LIN {X 0,Y 284.997,Z 899.013,A -85,B 0,C 180,E1 -17446.451,E2 -17446.451} C_VEL
LIN {X 0,Y 283.143,Z 901.991,A -85,B 0,C 180,E1 -17448.547,E2 -17448.547} C_VEL
LIN {X 0,Y 282.042,Z 903.588,A -85,B 0,C 180,E1 -17449.955,E2 -17449.955} C_VEL
LIN {X 0,Y 280.982,Z 904.651,A -85,B 0,C 180,E1 -17451.369,E2 -17451.369} C_VEL
LIN {X 0,Y 279.65,Z 905.657,A -85,B 0,C 180,E1 -17454.231,E2 -17454.231} C_VEL
LIN {X 0,Y 278.605,Z 905.018,A -85,B 0,C 180,E1 -17457.108,E2 -17457.108} C_VEL
LIN {X 0,Y 278.2,Z 904.125,A -85,B 0,C 180,E1 -17458.552,E2 -17458.552} C_VEL
LIN {X 0,Y 277.742,Z 902.734,A -85,B 0,C 180,E1 -17460,E2 -17460} C_VEL
LIN {X 0,Y 277.629,Z 899.945,A -85,B 0,C 180,E1 -17462.176,E2 -17462.176} C_VEL
LIN {X 0,Y 277.371,Z 896.204,A -85,B 0,C 180,E1 -17464.36,E2 -17464.36} C_VEL
LIN {X 0,Y 277.84,Z 891.35,A -85,B 0,C 180,E1 -17466.536,E2 -17466.536} C_VEL
LIN {X 0,Y 278.22,Z 885.341,A -85,B 0,C 180,E1 -17468.718,E2 -17468.718} C_VEL
LIN {X 0,Y 278.889,Z 876.721,A -85,B 0,C 180,E1 -17471.226,E2 -17471.226} C_VEL
LIN {X 0,Y 279.577,Z 868.835,A -85,B 0,C 180,E1 -17473.076,E2 -17473.076} C_VEL
LIN {X 0,Y 280.358,Z 859.638,A -85,B 0,C 180,E1 -17474.889,E2 -17474.889} C_VEL
LIN {X 0,Y 281.096,Z 850.958,A -85,B 0,C 180,E1 -17476.336,E2 -17476.336} C_VEL
LIN {X 0,Y 282.024,Z 840.057,A -85,B 0,C 180,E1 -17477.875,E2 -17477.875} C_VEL
LIN {X 0,Y 281.926,Z 836.631,A -85,B 0,C 180,E1 -17478.309,E2 -17478.309} C_VEL
LIN {X 0,Y 278.815,Z 824.242,A -85,B 0,C 180,E1 -17479.779,E2 -17479.779} C_VEL
LIN {X 0,Y 277.294,Z 817.935,A -85,B 0,C 180,E1 -17480.464,E2 -17480.464} C_VEL
LIN {X 0,Y 277.243,Z 817.949,A -85,B 0,C 180,E1 -17484.131,E2 -17484.131} C_VEL
LIN {X 0,Y 277.242,Z 817.938,A -85,B 0,C 180,E1 -17487.468,E2 -17487.468} C_VEL
LIN {X 0,Y 277.236,Z 817.947,A -85,B 0,C 180,E1 -17490.465,E2 -17490.465} C_VEL
LIN {X 0,Y 277.253,Z 817.94,A -85,B 0,C 180,E1 -17493.895,E2 -17493.895} C_VEL
LIN {X 0,Y 277.258,Z 817.939,A -85,B 0,C 180,E1 -17497.471,E2 -17497.471} C_VEL
LIN {X 0,Y 277.191,Z 817.953,A -85,B 0,C 180,E1 -17501.24,E2 -17501.24} C_VEL
LIN {X 0,Y 277.181,Z 817.956,A -85,B 0,C 180,E1 -17505.231,E2 -17505.231} C_VEL
LIN {X 0,Y 277.184,Z 817.956,A -85,B 0,C 180,E1 -17508.756,E2 -17508.756} C_VEL
LIN {X 0,Y 277.255,Z 817.945,A -85,B 0,C 180,E1 -17512.526,E2 -17512.526} C_VEL
LIN {X 0,Y 277.253,Z 817.95,A -85,B 0,C 180,E1 -17516.103,E2 -17516.103} C_VEL
LIN {X 0,Y 277.268,Z 817.941,A -85,B 0,C 180,E1 -17519.537,E2 -17519.537} C_VEL
LIN {X 0,Y 277.349,Z 817.93,A -85,B 0,C 180,E1 -17523.673,E2 -17523.673} C_VEL
LIN {X 0,Y 277.358,Z 817.943,A -85,B 0,C 180,E1 -17524.356,E2 -17524.356} C_VEL
LIN {X 0,Y 278.289,Z 820.641,A -85,B 0,C 180,E1 -17524.651,E2 -17524.651} C_VEL
LIN {X 0,Y 282.727,Z 831.715,A -85,B 0,C 180,E1 -17526.103,E2 -17526.103} C_VEL
LIN {X 0,Y 285.992,Z 841.823,A -85,B 0,C 180,E1 -17527.586,E2 -17527.586} C_VEL
LIN {X 0,Y 287.967,Z 848.891,A -85,B 0,C 180,E1 -17528.746,E2 -17528.746} C_VEL
LIN {X 0,Y 287.007,Z 857.045,A -85,B 0,C 180,E1 -17529.949,E2 -17529.949} C_VEL
LIN {X 0,Y 285.466,Z 866.858,A -85,B 0,C 180,E1 -17531.703,E2 -17531.703} C_VEL
LIN {X 0,Y 283.92,Z 874.9,A -85,B 0,C 180,E1 -17533.459,E2 -17533.459} C_VEL
LIN {X 0,Y 282.324,Z 882.758,A -85,B 0,C 180,E1 -17535.583,E2 -17535.583} C_VEL
LIN {X 0,Y 281.178,Z 889.027,A -85,B 0,C 180,E1 -17537.731,E2 -17537.731} C_VEL
LIN {X 0,Y 280.049,Z 894.02,A -85,B 0,C 180,E1 -17539.88,E2 -17539.88} C_VEL
LIN {X 0,Y 278.971,Z 897.914,A -85,B 0,C 180,E1 -17542.033,E2 -17542.033} C_VEL
LIN {X 0,Y 278.316,Z 900.764,A -85,B 0,C 180,E1 -17544.2,E2 -17544.2} C_VEL
LIN {X 0,Y 278.247,Z 902.093,A -85,B 0,C 180,E1 -17545.652,E2 -17545.652} C_VEL
LIN {X 0,Y 277.82,Z 903.673,A -85,B 0,C 180,E1 -17548.548,E2 -17548.548} C_VEL
LIN {X 0,Y 277.759,Z 903.902,A -85,B 0,C 180,E1 -17549.997,E2 -17549.997} C_VEL
LIN {X 0,Y 278.009,Z 903.133,A -85,B 0,C 180,E1 -17552.895,E2 -17552.895} C_VEL
LIN {X 0,Y 278.229,Z 902.189,A -85,B 0,C 180,E1 -17554.343,E2 -17554.343} C_VEL
LIN {X 0,Y 278.302,Z 900.9,A -85,B 0,C 180,E1 -17555.795,E2 -17555.795} C_VEL
LIN {X 0,Y 278.957,Z 898.092,A -85,B 0,C 180,E1 -17557.962,E2 -17557.962} C_VEL
LIN {X 0,Y 280.065,Z 894.248,A -85,B 0,C 180,E1 -17560.114,E2 -17560.114} C_VEL
LIN {X 0,Y 281.138,Z 889.336,A -85,B 0,C 180,E1 -17562.265,E2 -17562.265} C_VEL
LIN {X 0,Y 282.293,Z 883.16,A -85,B 0,C 180,E1 -17564.413,E2 -17564.413} C_VEL
LIN {X 0,Y 283.869,Z 875.385,A -85,B 0,C 180,E1 -17566.539,E2 -17566.539} C_VEL
LIN {X 0,Y 285.315,Z 867.455,A -85,B 0,C 180,E1 -17568.301,E2 -17568.301} C_VEL
LIN {X 0,Y 286.932,Z 857.756,A -85,B 0,C 180,E1 -17570.051,E2 -17570.051} C_VEL
LIN {X 0,Y 288.057,Z 849.407,A -85,B 0,C 180,E1 -17571.287,E2 -17571.287} C_VEL
LIN {X 0,Y 285.703,Z 840.645,A -85,B 0,C 180,E1 -17572.712,E2 -17572.712} C_VEL
LIN {X 0,Y 282.328,Z 830.734,A -85,B 0,C 180,E1 -17574.161,E2 -17574.161} C_VEL
LIN {X 0,Y 278.161,Z 820.468,A -85,B 0,C 180,E1 -17575.5,E2 -17575.5} C_VEL
LIN {X 0,Y 277.347,Z 817.939,A -85,B 0,C 180,E1 -17575.816,E2 -17575.816} C_VEL
LIN {X 0,Y 277.284,Z 817.946,A -85,B 0,C 180,E1 -17578.785,E2 -17578.785} C_VEL
LIN {X 0,Y 277.249,Z 817.95,A -85,B 0,C 180,E1 -17583.225,E2 -17583.225} C_VEL
LIN {X 0,Y 277.319,Z 817.944,A -85,B 0,C 180,E1 -17585.809,E2 -17585.809} C_VEL
LIN {X 0,Y 277.26,Z 817.948,A -85,B 0,C 180,E1 -17589.32,E2 -17589.32} C_VEL
LIN {X 0,Y 277.277,Z 817.945,A -85,B 0,C 180,E1 -17593.181,E2 -17593.181} C_VEL
LIN {X 0,Y 277.271,Z 817.939,A -85,B 0,C 180,E1 -17597.308,E2 -17597.308} C_VEL
LIN {X 0,Y 277.267,Z 817.942,A -85,B 0,C 180,E1 -17600.677,E2 -17600.677} C_VEL
LIN {X 0,Y 277.294,Z 817.943,A -85,B 0,C 180,E1 -17604.343,E2 -17604.343} C_VEL
LIN {X 0,Y 277.232,Z 817.95,A -85,B 0,C 180,E1 -17607.835,E2 -17607.835} C_VEL
LIN {X 0,Y 277.276,Z 817.946,A -85,B 0,C 180,E1 -17611.211,E2 -17611.211} C_VEL
LIN {X 0,Y 277.3,Z 817.937,A -85,B 0,C 180,E1 -17614.478,E2 -17614.478} C_VEL
LIN {X 0,Y 277.271,Z 817.944,A -85,B 0,C 180,E1 -17617.653,E2 -17617.653} C_VEL
LIN {X 0,Y 277.33,Z 817.937,A -85,B 0,C 180,E1 -17620.765,E2 -17620.765} C_VEL
LIN {X 0,Y 277.42,Z 817.92,A -85,B 0,C 180,E1 -17625.325,E2 -17625.325} C_VEL
LIN {X 0,Y 277.492,Z 817.914,A -85,B 0,C 180,E1 -17629.788,E2 -17629.788} C_VEL
LIN {X 0,Y 277.633,Z 817.902,A -85,B 0,C 180,E1 -17632.728,E2 -17632.728} C_VEL
LIN {X 0,Y 277.806,Z 817.881,A -85,B 0,C 180,E1 -17638.55,E2 -17638.55} C_VEL
LIN {X 0,Y 277.805,Z 817.884,A -85,B 0,C 180,E1 -17641.45,E2 -17641.45} C_VEL
LIN {X 0,Y 277.624,Z 817.903,A -85,B 0,C 180,E1 -17647.272,E2 -17647.272} C_VEL
LIN {X 0,Y 277.607,Z 817.904,A -85,B 0,C 180,E1 -17649.053,E2 -17649.053} C_VEL
LIN {X 0,Y 276.969,Z 817.986,A -85,B 0,C 180,E1 -17650.262,E2 -17650.262} C_VEL
LIN {X 0,Y 274.06,Z 818.349,A -85,B 0,C 180,E1 -17652.228,E2 -17652.228} C_VEL
LIN {X 0,Y 271.554,Z 818.659,A -85,B 0,C 180,E1 -17653.826,E2 -17653.826} C_VEL
LIN {X 0,Y 270.464,Z 818.795,A -85,B 0,C 180,E1 -17655.068,E2 -17655.068} C_VEL
LIN {X 0,Y 270.369,Z 818.807,A -85,B 0,C 180,E1 -17655.489,E2 -17655.489} C_VEL
LIN {X 0,Y 270.285,Z 818.819,A -85,B 0,C 180,E1 -17659.757,E2 -17659.757} C_VEL
LIN {X 0,Y 270.209,Z 818.826,A -85,B 0,C 180,E1 -17664.592,E2 -17664.592} C_VEL
LIN {X 0,Y 270.184,Z 818.825,A -85,B 0,C 180,E1 -17667.918,E2 -17667.918} C_VEL
LIN {X 0,Y 270.16,Z 818.833,A -85,B 0,C 180,E1 -17671.351,E2 -17671.351} C_VEL
LIN {X 0,Y 270.211,Z 818.827,A -85,B 0,C 180,E1 -17675.588,E2 -17675.588} C_VEL
LIN {X 0,Y 270.226,Z 818.92,A -85,B 0,C 180,E1 -17676.275,E2 -17676.275} C_VEL
LIN {X 0,Y 271.583,Z 825.509,A -85,B 0,C 180,E1 -17680.312,E2 -17680.312} C_VEL
LIN {X 0,Y 272.964,Z 832.072,A -85,B 0,C 180,E1 -17684.041,E2 -17684.041} C_VEL
LIN {X 0,Y 274.469,Z 840.068,A -85,B 0,C 180,E1 -17688.264,E2 -17688.264} C_VEL
LIN {X 0,Y 275.333,Z 845.207,A -85,B 0,C 180,E1 -17690.824,E2 -17690.824} C_VEL
LIN {X 0,Y 274.944,Z 848.645,A -85,B 0,C 180,E1 -17692.411,E2 -17692.411} C_VEL
LIN {X 0,Y 273.277,Z 857.605,A -85,B 0,C 180,E1 -17696.436,E2 -17696.436} C_VEL
LIN {X 0,Y 271.582,Z 868.258,A -85,B 0,C 180,E1 -17701.195,E2 -17701.195} C_VEL
LIN {X 0,Y 271.138,Z 871.591,A -85,B 0,C 180,E1 -17702.697,E2 -17702.697} C_VEL
LIN {X 0,Y 273.513,Z 886.239,A -85,B 0,C 180,E1 -17703.606,E2 -17703.606} C_VEL
LIN {X 0,Y 274.931,Z 899.031,A -85,B 0,C 180,E1 -17704.641,E2 -17704.641} C_VEL
LIN {X 0,Y 275.523,Z 911.781,A -85,B 0,C 180,E1 -17705.916,E2 -17705.916} C_VEL
LIN {X 0,Y 275.466,Z 923.215,A -85,B 0,C 180,E1 -17707.312,E2 -17707.312} C_VEL
LIN {X 0,Y 274.898,Z 933.568,A -85,B 0,C 180,E1 -17708.834,E2 -17708.834} C_VEL
LIN {X 0,Y 274.438,Z 941.169,A -85,B 0,C 180,E1 -17710.168,E2 -17710.168} C_VEL
LIN {X 0,Y 272.711,Z 950.162,A -85,B 0,C 180,E1 -17711.989,E2 -17711.989} C_VEL
LIN {X 0,Y 271.023,Z 958.971,A -85,B 0,C 180,E1 -17714.203,E2 -17714.203} C_VEL
LIN {X 0,Y 270.056,Z 966.097,A -85,B 0,C 180,E1 -17716.457,E2 -17716.457} C_VEL
LIN {X 0,Y 269.414,Z 971.84,A -85,B 0,C 180,E1 -17718.72,E2 -17718.72} C_VEL
LIN {X 0,Y 269.186,Z 976.397,A -85,B 0,C 180,E1 -17720.99,E2 -17720.99} C_VEL
LIN {X 0,Y 269.222,Z 979.193,A -85,B 0,C 180,E1 -17722.741,E2 -17722.741} C_VEL
LIN {X 0,Y 269.55,Z 982.334,A -85,B 0,C 180,E1 -17725.517,E2 -17725.517} C_VEL
LIN {X 0,Y 269.706,Z 983.411,A -85,B 0,C 180,E1 -17727.015,E2 -17727.015} C_VEL
LIN {X 0,Y 269.852,Z 984.074,A -85,B 0,C 180,E1 -17728.51,E2 -17728.51} C_VEL
LIN {X 0,Y 269.995,Z 984.319,A -85,B 0,C 180,E1 -17730.003,E2 -17730.003} C_VEL
LIN {X 0,Y 269.853,Z 984.064,A -85,B 0,C 180,E1 -17731.495,E2 -17731.495} C_VEL
LIN {X 0,Y 269.71,Z 983.395,A -85,B 0,C 180,E1 -17732.99,E2 -17732.99} C_VEL
LIN {X 0,Y 269.575,Z 982.315,A -85,B 0,C 180,E1 -17734.488,E2 -17734.488} C_VEL
LIN {X 0,Y 269.238,Z 979.122,A -85,B 0,C 180,E1 -17737.284,E2 -17737.284} C_VEL
LIN {X 0,Y 269.529,Z 971.343,A -85,B 0,C 180,E1 -17742.043,E2 -17742.043} C_VEL
LIN {X 0,Y 270.381,Z 966.739,A -85,B 0,C 180,E1 -17744.299,E2 -17744.299} C_VEL
LIN {X 0,Y 271.681,Z 961.017,A -85,B 0,C 180,E1 -17746.535,E2 -17746.535} C_VEL
LIN {X 0,Y 273.549,Z 954.239,A -85,B 0,C 180,E1 -17748.735,E2 -17748.735} C_VEL
LIN {X 0,Y 275.991,Z 946.224,A -85,B 0,C 180,E1 -17750.888,E2 -17750.888} C_VEL
LIN {X 0,Y 277.399,Z 940.261,A -85,B 0,C 180,E1 -17752.338,E2 -17752.338} C_VEL
LIN {X 0,Y 279.567,Z 929.919,A -85,B 0,C 180,E1 -17754.509,E2 -17754.509} C_VEL
LIN {X 0,Y 281.86,Z 919.067,A -85,B 0,C 180,E1 -17756.455,E2 -17756.455} C_VEL
LIN {X 0,Y 282.915,Z 909.244,A -85,B 0,C 180,E1 -17758.166,E2 -17758.166} C_VEL
LIN {X 0,Y 283.359,Z 896.995,A -85,B 0,C 180,E1 -17760.265,E2 -17760.265} C_VEL
LIN {X 0,Y 283.177,Z 886.629,A -85,B 0,C 180,E1 -17762.084,E2 -17762.084} C_VEL
LIN {X 0,Y 282.457,Z 875.054,A -85,B 0,C 180,E1 -17764.252,E2 -17764.252} C_VEL
LIN {X 0,Y 281.688,Z 866.988,A -85,B 0,C 180,E1 -17765.899,E2 -17765.899} C_VEL
LIN {X 0,Y 281.166,Z 861.203,A -85,B 0,C 180,E1 -17767.187,E2 -17767.187} C_VEL
LIN {X 0,Y 281.146,Z 859.94,A -85,B 0,C 180,E1 -17767.42,E2 -17767.42} C_VEL
LIN {X 0,Y 279.903,Z 851.044,A -85,B 0,C 180,E1 -17769.942,E2 -17769.942} C_VEL
LIN {X 0,Y 279.125,Z 846.061,A -85,B 0,C 180,E1 -17771.937,E2 -17771.937} C_VEL
LIN {X 0,Y 278.623,Z 842.393,A -85,B 0,C 180,E1 -17773.993,E2 -17773.993} C_VEL
LIN {X 0,Y 278.659,Z 839.748,A -85,B 0,C 180,E1 -17776.004,E2 -17776.004} C_VEL
LIN {X 0,Y 278.898,Z 838.691,A -85,B 0,C 180,E1 -17777.127,E2 -17777.127} C_VEL
LIN {X 0,Y 279.657,Z 837.646,A -85,B 0,C 180,E1 -17779.201,E2 -17779.201} C_VEL
LIN {X 0,Y 280.989,Z 837.503,A -85,B 0,C 180,E1 -17781.296,E2 -17781.296} C_VEL
LIN {X 0,Y 282.724,Z 838.756,A -85,B 0,C 180,E1 -17783.373,E2 -17783.373} C_VEL
LIN {X 0,Y 284.775,Z 840.777,A -85,B 0,C 180,E1 -17785.415,E2 -17785.415} C_VEL
LIN {X 0,Y 287.225,Z 843.725,A -85,B 0,C 180,E1 -17787.431,E2 -17787.431} C_VEL
LIN {X 0,Y 290.331,Z 851.625,A -85,B 0,C 180,E1 -17790.631,E2 -17790.631} C_VEL
LIN {X 0,Y 292.153,Z 858.072,A -85,B 0,C 180,E1 -17792.802,E2 -17792.802} C_VEL
LIN {X 0,Y 293.327,Z 864.655,A -85,B 0,C 180,E1 -17794.831,E2 -17794.831} C_VEL
LIN {X 0,Y 293.448,Z 865.932,A -85,B 0,C 180,E1 -17795.221,E2 -17795.221} C_VEL
LIN {X 0,Y 291.978,Z 870.915,A -85,B 0,C 180,E1 -17796.185,E2 -17796.185} C_VEL
LIN {X 0,Y 288.671,Z 879.706,A -85,B 0,C 180,E1 -17798.129,E2 -17798.129} C_VEL
LIN {X 0,Y 285.979,Z 886.069,A -85,B 0,C 180,E1 -17799.876,E2 -17799.876} C_VEL
LIN {X 0,Y 284.047,Z 890.377,A -85,B 0,C 180,E1 -17801.237,E2 -17801.237} C_VEL
LIN {X 0,Y 281.48,Z 895.633,A -85,B 0,C 180,E1 -17803.314,E2 -17803.314} C_VEL
LIN {X 0,Y 279.135,Z 899.868,A -85,B 0,C 180,E1 -17805.417,E2 -17805.417} C_VEL
LIN {X 0,Y 277.722,Z 902.115,A -85,B 0,C 180,E1 -17806.835,E2 -17806.835} C_VEL
LIN {X 0,Y 275.261,Z 905.236,A -85,B 0,C 180,E1 -17809.705,E2 -17809.705} C_VEL
LIN {X 0,Y 274.166,Z 906.273,A -85,B 0,C 180,E1 -17811.153,E2 -17811.153} C_VEL
LIN {X 0,Y 272.71,Z 906.976,A -85,B 0,C 180,E1 -17814.083,E2 -17814.083} C_VEL
LIN {X 0,Y 272.154,Z 906.742,A -85,B 0,C 180,E1 -17815.557,E2 -17815.557} C_VEL
LIN {X 0,Y 271.615,Z 906.142,A -85,B 0,C 180,E1 -17817.034,E2 -17817.034} C_VEL
LIN {X 0,Y 271.188,Z 905.089,A -85,B 0,C 180,E1 -17818.515,E2 -17818.515} C_VEL
LIN {X 0,Y 270.715,Z 903.642,A -85,B 0,C 180,E1 -17820,E2 -17820} C_VEL
LIN {X 0,Y 270.594,Z 900.68,A -85,B 0,C 180,E1 -17822.233,E2 -17822.233} C_VEL
LIN {X 0,Y 270.333,Z 896.764,A -85,B 0,C 180,E1 -17824.473,E2 -17824.473} C_VEL
LIN {X 0,Y 270.798,Z 891.735,A -85,B 0,C 180,E1 -17826.707,E2 -17826.707} C_VEL
LIN {X 0,Y 271.322,Z 883.824,A -85,B 0,C 180,E1 -17829.462,E2 -17829.462} C_VEL
LIN {X 0,Y 271.916,Z 876.431,A -85,B 0,C 180,E1 -17831.555,E2 -17831.555} C_VEL
LIN {X 0,Y 272.631,Z 868.408,A -85,B 0,C 180,E1 -17833.415,E2 -17833.415} C_VEL
LIN {X 0,Y 273.356,Z 859.973,A -85,B 0,C 180,E1 -17835.089,E2 -17835.089} C_VEL
LIN {X 0,Y 274.112,Z 851.176,A -85,B 0,C 180,E1 -17836.573,E2 -17836.573} C_VEL
LIN {X 0,Y 275.005,Z 840.836,A -85,B 0,C 180,E1 -17838.057,E2 -17838.057} C_VEL
LIN {X 0,Y 275.02,Z 838.204,A -85,B 0,C 180,E1 -17838.396,E2 -17838.396} C_VEL
LIN {X 0,Y 271.851,Z 825.586,A -85,B 0,C 180,E1 -17839.946,E2 -17839.946} C_VEL
LIN {X 0,Y 270.24,Z 818.813,A -85,B 0,C 180,E1 -17840.679,E2 -17840.679} C_VEL
LIN {X 0,Y 270.185,Z 818.827,A -85,B 0,C 180,E1 -17844.594,E2 -17844.594} C_VEL
LIN {X 0,Y 270.192,Z 818.818,A -85,B 0,C 180,E1 -17847.918,E2 -17847.918} C_VEL
LIN {X 0,Y 270.177,Z 818.826,A -85,B 0,C 180,E1 -17851.349,E2 -17851.349} C_VEL
LIN {X 0,Y 270.205,Z 818.823,A -85,B 0,C 180,E1 -17854.905,E2 -17854.905} C_VEL
LIN {X 0,Y 270.206,Z 818.822,A -85,B 0,C 180,E1 -17858.709,E2 -17858.709} C_VEL
LIN {X 0,Y 270.156,Z 818.828,A -85,B 0,C 180,E1 -17863.244,E2 -17863.244} C_VEL
LIN {X 0,Y 270.158,Z 818.83,A -85,B 0,C 180,E1 -17867.436,E2 -17867.436} C_VEL
LIN {X 0,Y 270.173,Z 818.831,A -85,B 0,C 180,E1 -17871.366,E2 -17871.366} C_VEL
LIN {X 0,Y 270.205,Z 818.825,A -85,B 0,C 180,E1 -17875.092,E2 -17875.092} C_VEL
LIN {X 0,Y 270.207,Z 818.82,A -85,B 0,C 180,E1 -17879.129,E2 -17879.129} C_VEL
LIN {X 0,Y 270.307,Z 818.807,A -85,B 0,C 180,E1 -17883.61,E2 -17883.61} C_VEL
LIN {X 0,Y 270.881,Z 820.853,A -85,B 0,C 180,E1 -17883.826,E2 -17883.826} C_VEL
LIN {X 0,Y 275.054,Z 830.761,A -85,B 0,C 180,E1 -17885.164,E2 -17885.164} C_VEL
LIN {X 0,Y 278.475,Z 840.628,A -85,B 0,C 180,E1 -17886.638,E2 -17886.638} C_VEL
LIN {X 0,Y 281.211,Z 850.251,A -85,B 0,C 180,E1 -17888.255,E2 -17888.255} C_VEL
LIN {X 0,Y 281.158,Z 853.471,A -85,B 0,C 180,E1 -17888.749,E2 -17888.749} C_VEL
LIN {X 0,Y 279.711,Z 862.284,A -85,B 0,C 180,E1 -17890.169,E2 -17890.169} C_VEL
LIN {X 0,Y 278.168,Z 871.306,A -85,B 0,C 180,E1 -17891.968,E2 -17891.968} C_VEL
LIN {X 0,Y 276.276,Z 880.085,A -85,B 0,C 180,E1 -17894.127,E2 -17894.127} C_VEL
LIN {X 0,Y 274.95,Z 886.884,A -85,B 0,C 180,E1 -17896.246,E2 -17896.246} C_VEL
LIN {X 0,Y 273.976,Z 891.821,A -85,B 0,C 180,E1 -17898.155,E2 -17898.155} C_VEL
LIN {X 0,Y 272.659,Z 896.459,A -85,B 0,C 180,E1 -17900.352,E2 -17900.352} C_VEL
LIN {X 0,Y 271.763,Z 899.981,A -85,B 0,C 180,E1 -17902.568,E2 -17902.568} C_VEL
LIN {X 0,Y 271.328,Z 901.796,A -85,B 0,C 180,E1 -17904.05,E2 -17904.05} C_VEL
LIN {X 0,Y 271.244,Z 903.125,A -85,B 0,C 180,E1 -17905.539,E2 -17905.539} C_VEL
LIN {X 0,Y 270.798,Z 904.704,A -85,B 0,C 180,E1 -17908.51,E2 -17908.51} C_VEL
LIN {X 0,Y 270.735,Z 904.933,A -85,B 0,C 180,E1 -17909.997,E2 -17909.997} C_VEL
LIN {X 0,Y 270.995,Z 904.163,A -85,B 0,C 180,E1 -17912.97,E2 -17912.97} C_VEL
LIN {X 0,Y 271.228,Z 903.22,A -85,B 0,C 180,E1 -17914.456,E2 -17914.456} C_VEL
LIN {X 0,Y 271.314,Z 901.93,A -85,B 0,C 180,E1 -17915.945,E2 -17915.945} C_VEL
LIN {X 0,Y 272.002,Z 899.123,A -85,B 0,C 180,E1 -17918.167,E2 -17918.167} C_VEL
LIN {X 0,Y 273.152,Z 895.278,A -85,B 0,C 180,E1 -17920.373,E2 -17920.373} C_VEL
LIN {X 0,Y 274.281,Z 890.365,A -85,B 0,C 180,E1 -17922.577,E2 -17922.577} C_VEL
LIN {X 0,Y 275.496,Z 884.189,A -85,B 0,C 180,E1 -17924.777,E2 -17924.777} C_VEL
LIN {X 0,Y 277.142,Z 876.414,A -85,B 0,C 180,E1 -17926.952,E2 -17926.952} C_VEL
LIN {X 0,Y 278.666,Z 868.481,A -85,B 0,C 180,E1 -17928.754,E2 -17928.754} C_VEL
LIN {X 0,Y 280.349,Z 858.783,A -85,B 0,C 180,E1 -17930.543,E2 -17930.543} C_VEL
LIN {X 0,Y 281.375,Z 852.217,A -85,B 0,C 180,E1 -17931.545,E2 -17931.545} C_VEL
LIN {X 0,Y 280.804,Z 848.504,A -85,B 0,C 180,E1 -17932.174,E2 -17932.174} C_VEL
LIN {X 0,Y 277.633,Z 837.999,A -85,B 0,C 180,E1 -17933.889,E2 -17933.889} C_VEL
LIN {X 0,Y 273.945,Z 827.91,A -85,B 0,C 180,E1 -17935.351,E2 -17935.351} C_VEL
LIN {X 0,Y 270.36,Z 819.221,A -85,B 0,C 180,E1 -17936.476,E2 -17936.476} C_VEL
LIN {X 0,Y 270.304,Z 818.816,A -85,B 0,C 180,E1 -17936.54,E2 -17936.54} C_VEL
LIN {X 0,Y 270.195,Z 818.829,A -85,B 0,C 180,E1 -17940.867,E2 -17940.867} C_VEL
LIN {X 0,Y 270.209,Z 818.827,A -85,B 0,C 180,E1 -17944.901,E2 -17944.901} C_VEL
LIN {X 0,Y 270.214,Z 818.827,A -85,B 0,C 180,E1 -17948.714,E2 -17948.714} C_VEL
LIN {X 0,Y 270.253,Z 818.822,A -85,B 0,C 180,E1 -17952.538,E2 -17952.538} C_VEL
LIN {X 0,Y 270.223,Z 818.82,A -85,B 0,C 180,E1 -17956.733,E2 -17956.733} C_VEL
LIN {X 0,Y 270.254,Z 818.82,A -85,B 0,C 180,E1 -17959.448,E2 -17959.448} C_VEL
LIN {X 0,Y 270.247,Z 818.82,A -85,B 0,C 180,E1 -17963.719,E2 -17963.719} C_VEL
LIN {X 0,Y 270.192,Z 818.828,A -85,B 0,C 180,E1 -17966.891,E2 -17966.891} C_VEL
LIN {X 0,Y 270.216,Z 818.819,A -85,B 0,C 180,E1 -17970.385,E2 -17970.385} C_VEL
LIN {X 0,Y 270.25,Z 818.816,A -85,B 0,C 180,E1 -17973.762,E2 -17973.762} C_VEL
LIN {X 0,Y 270.219,Z 818.826,A -85,B 0,C 180,E1 -17977.037,E2 -17977.037} C_VEL
LIN {X 0,Y 270.287,Z 818.812,A -85,B 0,C 180,E1 -17980.243,E2 -17980.243} C_VEL
LIN {X 0,Y 270.388,Z 818.794,A -85,B 0,C 180,E1 -17984.934,E2 -17984.934} C_VEL
LIN {X 0,Y 270.427,Z 818.795,A -85,B 0,C 180,E1 -17989.518,E2 -17989.518} C_VEL
LIN {X 0,Y 270.592,Z 818.778,A -85,B 0,C 180,E1 -17992.538,E2 -17992.538} C_VEL
LIN {X 0,Y 270.772,Z 818.758,A -85,B 0,C 180,E1 -17998.513,E2 -17998.513} C_VEL
LIN {X 0,Y 270.77,Z 818.761,A -85,B 0,C 180,E1 -18001.487,E2 -18001.487} C_VEL
LIN {X 0,Y 270.584,Z 818.781,A -85,B 0,C 180,E1 -18007.462,E2 -18007.462} C_VEL
LIN {X 0,Y 270.426,Z 818.798,A -85,B 0,C 180,E1 -18010.482,E2 -18010.482} C_VEL
LIN {X 0,Y 270.369,Z 818.807,A -85,B 0,C 180,E1 -18015.489,E2 -18015.489} C_VEL
LIN {X 0,Y 269.677,Z 818.896,A -85,B 0,C 180,E1 -18016.731,E2 -18016.731} C_VEL
LIN {X 0,Y 266.778,Z 819.263,A -85,B 0,C 180,E1 -18018.753,E2 -18018.753} C_VEL
LIN {X 0,Y 264.307,Z 819.571,A -85,B 0,C 180,E1 -18020.397,E2 -18020.397} C_VEL
LIN {X 0,Y 263.221,Z 819.701,A -85,B 0,C 180,E1 -18021.673,E2 -18021.673} C_VEL
LIN {X 0,Y 263.118,Z 819.71,A -85,B 0,C 180,E1 -18022.106,E2 -18022.106} C_VEL
LIN {X 0,Y 263.153,Z 819.704,A -85,B 0,C 180,E1 -18025.297,E2 -18025.297} C_VEL
LIN {X 0,Y 263.119,Z 819.712,A -85,B 0,C 180,E1 -18028.737,E2 -18028.737} C_VEL
LIN {X 0,Y 263.114,Z 819.708,A -85,B 0,C 180,E1 -18032.291,E2 -18032.291} C_VEL
LIN {X 0,Y 263.196,Z 819.769,A -85,B 0,C 180,E1 -18035.506,E2 -18035.506} C_VEL
LIN {X 0,Y 264.498,Z 826.24,A -85,B 0,C 180,E1 -18039.621,E2 -18039.621} C_VEL
LIN {X 0,Y 265.833,Z 832.682,A -85,B 0,C 180,E1 -18043.423,E2 -18043.423} C_VEL
LIN {X 0,Y 267.239,Z 840.004,A -85,B 0,C 180,E1 -18047.422,E2 -18047.422} C_VEL
LIN {X 0,Y 268.223,Z 845.529,A -85,B 0,C 180,E1 -18050.307,E2 -18050.307} C_VEL
LIN {X 0,Y 268.367,Z 847.054,A -85,B 0,C 180,E1 -18051.064,E2 -18051.064} C_VEL
LIN {X 0,Y 266.939,Z 854.856,A -85,B 0,C 180,E1 -18054.704,E2 -18054.704} C_VEL
LIN {X 0,Y 264.953,Z 865.764,A -85,B 0,C 180,E1 -18059.74,E2 -18059.74} C_VEL
LIN {X 0,Y 264.257,Z 870.498,A -85,B 0,C 180,E1 -18061.93,E2 -18061.93} C_VEL
LIN {X 0,Y 266.677,Z 885.004,A -85,B 0,C 180,E1 -18062.868,E2 -18062.868} C_VEL
LIN {X 0,Y 268.111,Z 897.835,A -85,B 0,C 180,E1 -18063.94,E2 -18063.94} C_VEL
LIN {X 0,Y 268.753,Z 910.695,A -85,B 0,C 180,E1 -18065.269,E2 -18065.269} C_VEL
LIN {X 0,Y 268.708,Z 922.178,A -85,B 0,C 180,E1 -18066.714,E2 -18066.714} C_VEL
LIN {X 0,Y 268.014,Z 933.671,A -85,B 0,C 180,E1 -18068.465,E2 -18068.465} C_VEL
LIN {X 0,Y 267.698,Z 940.118,A -85,B 0,C 180,E1 -18069.647,E2 -18069.647} C_VEL
LIN {X 0,Y 265.912,Z 949.113,A -85,B 0,C 180,E1 -18071.512,E2 -18071.512} C_VEL
LIN {X 0,Y 264.357,Z 956.309,A -85,B 0,C 180,E1 -18073.327,E2 -18073.327} C_VEL
LIN {X 0,Y 263.255,Z 963.986,A -85,B 0,C 180,E1 -18075.706,E2 -18075.706} C_VEL
LIN {X 0,Y 262.561,Z 969.018,A -85,B 0,C 180,E1 -18077.638,E2 -18077.638} C_VEL
LIN {X 0,Y 262.171,Z 973.962,A -85,B 0,C 180,E1 -18079.968,E2 -18079.968} C_VEL
LIN {X 0,Y 262.157,Z 978.368,A -85,B 0,C 180,E1 -18082.708,E2 -18082.708} C_VEL
LIN {X 0,Y 262.472,Z 981.292,A -85,B 0,C 180,E1 -18085.395,E2 -18085.395} C_VEL
LIN {X 0,Y 262.652,Z 982.374,A -85,B 0,C 180,E1 -18086.935,E2 -18086.935} C_VEL
LIN {X 0,Y 262.812,Z 983.04,A -85,B 0,C 180,E1 -18088.47,E2 -18088.47} C_VEL
LIN {X 0,Y 262.966,Z 983.287,A -85,B 0,C 180,E1 -18090.003,E2 -18090.003} C_VEL
LIN {X 0,Y 262.813,Z 983.03,A -85,B 0,C 180,E1 -18091.535,E2 -18091.535} C_VEL
LIN {X 0,Y 262.658,Z 982.358,A -85,B 0,C 180,E1 -18093.07,E2 -18093.07} C_VEL
LIN {X 0,Y 262.497,Z 981.272,A -85,B 0,C 180,E1 -18094.61,E2 -18094.61} C_VEL
LIN {X 0,Y 262.181,Z 978.285,A -85,B 0,C 180,E1 -18097.333,E2 -18097.333} C_VEL
LIN {X 0,Y 262.516,Z 970.743,A -85,B 0,C 180,E1 -18102.37,E2 -18102.37} C_VEL
LIN {X 0,Y 263.873,Z 964.582,A -85,B 0,C 180,E1 -18105.449,E2 -18105.449} C_VEL
LIN {X 0,Y 265.397,Z 958.852,A -85,B 0,C 180,E1 -18107.683,E2 -18107.683} C_VEL
LIN {X 0,Y 267.593,Z 951.843,A -85,B 0,C 180,E1 -18109.967,E2 -18109.967} C_VEL
LIN {X 0,Y 270.222,Z 943.76,A -85,B 0,C 180,E1 -18112.158,E2 -18112.158} C_VEL
LIN {X 0,Y 271.999,Z 936.185,A -85,B 0,C 180,E1 -18114.016,E2 -18114.016} C_VEL
LIN {X 0,Y 274.407,Z 926.326,A -85,B 0,C 180,E1 -18116.056,E2 -18116.056} C_VEL
LIN {X 0,Y 276.084,Z 918.79,A -85,B 0,C 180,E1 -18117.479,E2 -18117.479} C_VEL
LIN {X 0,Y 277.419,Z 907.351,A -85,B 0,C 180,E1 -18119.603,E2 -18119.603} C_VEL
LIN {X 0,Y 278.078,Z 895.309,A -85,B 0,C 180,E1 -18121.818,E2 -18121.818} C_VEL
LIN {X 0,Y 278.037,Z 883.915,A -85,B 0,C 180,E1 -18124.033,E2 -18124.033} C_VEL
LIN {X 0,Y 277.75,Z 872.13,A -85,B 0,C 180,E1 -18126.49,E2 -18126.49} C_VEL
LIN {X 0,Y 277.299,Z 863.226,A -85,B 0,C 180,E1 -18128.613,E2 -18128.613} C_VEL
LIN {X 0,Y 276.739,Z 855.799,A -85,B 0,C 180,E1 -18130.908,E2 -18130.908} C_VEL
LIN {X 0,Y 276.338,Z 852.031,A -85,B 0,C 180,E1 -18132.477,E2 -18132.477} C_VEL
LIN {X 0,Y 276.049,Z 848.521,A -85,B 0,C 180,E1 -18134.532,E2 -18134.532} C_VEL
LIN {X 0,Y 276.271,Z 845.928,A -85,B 0,C 180,E1 -18136.619,E2 -18136.619} C_VEL
LIN {X 0,Y 276.924,Z 844.556,A -85,B 0,C 180,E1 -18138.711,E2 -18138.711} C_VEL
LIN {X 0,Y 278.525,Z 844.174,A -85,B 0,C 180,E1 -18141.467,E2 -18141.467} C_VEL
LIN {X 0,Y 279.914,Z 845.341,A -85,B 0,C 180,E1 -18143.464,E2 -18143.464} C_VEL
LIN {X 0,Y 281.736,Z 847.264,A -85,B 0,C 180,E1 -18145.409,E2 -18145.409} C_VEL
LIN {X 0,Y 283.638,Z 850.115,A -85,B 0,C 180,E1 -18147.403,E2 -18147.403} C_VEL
LIN {X 0,Y 285.68,Z 856.242,A -85,B 0,C 180,E1 -18150.043,E2 -18150.043} C_VEL
LIN {X 0,Y 287.127,Z 862.353,A -85,B 0,C 180,E1 -18152.286,E2 -18152.286} C_VEL
LIN {X 0,Y 287.851,Z 867.27,A -85,B 0,C 180,E1 -18153.929,E2 -18153.929} C_VEL
LIN {X 0,Y 287.985,Z 869.2,A -85,B 0,C 180,E1 -18154.552,E2 -18154.552} C_VEL
LIN {X 0,Y 286.039,Z 874.712,A -85,B 0,C 180,E1 -18155.697,E2 -18155.697} C_VEL
LIN {X 0,Y 282.605,Z 883.085,A -85,B 0,C 180,E1 -18157.674,E2 -18157.674} C_VEL
LIN {X 0,Y 278.78,Z 891.138,A -85,B 0,C 180,E1 -18160.103,E2 -18160.103} C_VEL
LIN {X 0,Y 275.966,Z 896.516,A -85,B 0,C 180,E1 -18162.206,E2 -18162.206} C_VEL
LIN {X 0,Y 272.585,Z 902.015,A -85,B 0,C 180,E1 -18165.059,E2 -18165.059} C_VEL
LIN {X 0,Y 271.096,Z 904.076,A -85,B 0,C 180,E1 -18166.507,E2 -18166.507} C_VEL
LIN {X 0,Y 268.492,Z 906.902,A -85,B 0,C 180,E1 -18169.442,E2 -18169.442} C_VEL
LIN {X 0,Y 267.338,Z 907.846,A -85,B 0,C 180,E1 -18170.925,E2 -18170.925} C_VEL
LIN {X 0,Y 265.773,Z 908.296,A -85,B 0,C 180,E1 -18173.928,E2 -18173.928} C_VEL
LIN {X 0,Y 265.184,Z 907.958,A -85,B 0,C 180,E1 -18175.44,E2 -18175.44} C_VEL
LIN {X 0,Y 264.622,Z 907.198,A -85,B 0,C 180,E1 -18176.955,E2 -18176.955} C_VEL
LIN {X 0,Y 263.687,Z 904.529,A -85,B 0,C 180,E1 -18180,E2 -18180} C_VEL
LIN {X 0,Y 263.554,Z 901.389,A -85,B 0,C 180,E1 -18182.292,E2 -18182.292} C_VEL
LIN {X 0,Y 263.298,Z 897.281,A -85,B 0,C 180,E1 -18184.593,E2 -18184.593} C_VEL
LIN {X 0,Y 263.829,Z 890.99,A -85,B 0,C 180,E1 -18187.269,E2 -18187.269} C_VEL
LIN {X 0,Y 264.185,Z 885.539,A -85,B 0,C 180,E1 -18189.185,E2 -18189.185} C_VEL
LIN {X 0,Y 264.794,Z 877.661,A -85,B 0,C 180,E1 -18191.482,E2 -18191.482} C_VEL
LIN {X 0,Y 265.514,Z 869.659,A -85,B 0,C 180,E1 -18193.392,E2 -18193.392} C_VEL
LIN {X 0,Y 266.244,Z 861.253,A -85,B 0,C 180,E1 -18195.11,E2 -18195.11} C_VEL
LIN {X 0,Y 267.014,Z 852.496,A -85,B 0,C 180,E1 -18196.633,E2 -18196.633} C_VEL
LIN {X 0,Y 267.978,Z 842.292,A -85,B 0,C 180,E1 -18198.146,E2 -18198.146} C_VEL
LIN {X 0,Y 267.922,Z 838.94,A -85,B 0,C 180,E1 -18198.593,E2 -18198.593} C_VEL
LIN {X 0,Y 264.744,Z 826.155,A -85,B 0,C 180,E1 -18200.188,E2 -18200.188} C_VEL
LIN {X 0,Y 263.198,Z 819.689,A -85,B 0,C 180,E1 -18200.9,E2 -18200.9} C_VEL
LIN {X 0,Y 263.127,Z 819.707,A -85,B 0,C 180,E1 -18205.3,E2 -18205.3} C_VEL
LIN {X 0,Y 263.125,Z 819.702,A -85,B 0,C 180,E1 -18208.736,E2 -18208.736} C_VEL
LIN {X 0,Y 263.134,Z 819.694,A -85,B 0,C 180,E1 -18212.288,E2 -18212.288} C_VEL
LIN {X 0,Y 263.181,Z 819.694,A -85,B 0,C 180,E1 -18216.759,E2 -18216.759} C_VEL
LIN {X 0,Y 263.099,Z 819.711,A -85,B 0,C 180,E1 -18219.874,E2 -18219.874} C_VEL
LIN {X 0,Y 263.084,Z 819.714,A -85,B 0,C 180,E1 -18223.993,E2 -18223.993} C_VEL
LIN {X 0,Y 263.081,Z 819.715,A -85,B 0,C 180,E1 -18228.418,E2 -18228.418} C_VEL
LIN {X 0,Y 263.121,Z 819.709,A -85,B 0,C 180,E1 -18232.094,E2 -18232.094} C_VEL
LIN {X 0,Y 263.158,Z 819.704,A -85,B 0,C 180,E1 -18235.884,E2 -18235.884} C_VEL
LIN {X 0,Y 263.148,Z 819.7,A -85,B 0,C 180,E1 -18239.504,E2 -18239.504} C_VEL
LIN {X 0,Y 263.266,Z 819.682,A -85,B 0,C 180,E1 -18242.82,E2 -18242.82} C_VEL
LIN {X 0,Y 264.786,Z 823.715,A -85,B 0,C 180,E1 -18243.329,E2 -18243.329} C_VEL
LIN {X 0,Y 269.238,Z 834.657,A -85,B 0,C 180,E1 -18244.905,E2 -18244.905} C_VEL
LIN {X 0,Y 272.303,Z 843.946,A -85,B 0,C 180,E1 -18246.383,E2 -18246.383} C_VEL
LIN {X 0,Y 274.425,Z 851.617,A -85,B 0,C 180,E1 -18247.734,E2 -18247.734} C_VEL
LIN {X 0,Y 274.755,Z 853.614,A -85,B 0,C 180,E1 -18248.09,E2 -18248.09} C_VEL
LIN {X 0,Y 273.116,Z 863.318,A -85,B 0,C 180,E1 -18249.67,E2 -18249.67} C_VEL
LIN {X 0,Y 271.503,Z 872.339,A -85,B 0,C 180,E1 -18251.51,E2 -18251.51} C_VEL
LIN {X 0,Y 269.526,Z 881.119,A -85,B 0,C 180,E1 -18253.719,E2 -18253.719} C_VEL
LIN {X 0,Y 268.129,Z 887.918,A -85,B 0,C 180,E1 -18255.889,E2 -18255.889} C_VEL
LIN {X 0,Y 267.108,Z 892.854,A -85,B 0,C 180,E1 -18257.846,E2 -18257.846} C_VEL
LIN {X 0,Y 265.737,Z 897.491,A -85,B 0,C 180,E1 -18260.099,E2 -18260.099} C_VEL
LIN {X 0,Y 264.798,Z 901.013,A -85,B 0,C 180,E1 -18262.371,E2 -18262.371} C_VEL
LIN {X 0,Y 264.342,Z 902.828,A -85,B 0,C 180,E1 -18263.893,E2 -18263.893} C_VEL
LIN {X 0,Y 264.242,Z 904.157,A -85,B 0,C 180,E1 -18265.421,E2 -18265.421} C_VEL
LIN {X 0,Y 263.777,Z 905.736,A -85,B 0,C 180,E1 -18268.471,E2 -18268.471} C_VEL
LIN {X 0,Y 263.711,Z 905.965,A -85,B 0,C 180,E1 -18269.997,E2 -18269.997} C_VEL
LIN {X 0,Y 263.981,Z 905.194,A -85,B 0,C 180,E1 -18273.049,E2 -18273.049} C_VEL
LIN {X 0,Y 264.227,Z 904.25,A -85,B 0,C 180,E1 -18274.574,E2 -18274.574} C_VEL
LIN {X 0,Y 264.327,Z 902.961,A -85,B 0,C 180,E1 -18276.102,E2 -18276.102} C_VEL
LIN {X 0,Y 265.05,Z 900.153,A -85,B 0,C 180,E1 -18278.383,E2 -18278.383} C_VEL
LIN {X 0,Y 266.246,Z 896.308,A -85,B 0,C 180,E1 -18280.645,E2 -18280.645} C_VEL
LIN {X 0,Y 267.435,Z 891.394,A -85,B 0,C 180,E1 -18282.904,E2 -18282.904} C_VEL
LIN {X 0,Y 268.71,Z 885.218,A -85,B 0,C 180,E1 -18285.159,E2 -18285.159} C_VEL
LIN {X 0,Y 270.432,Z 877.443,A -85,B 0,C 180,E1 -18287.386,E2 -18287.386} C_VEL
LIN {X 0,Y 272.032,Z 869.508,A -85,B 0,C 180,E1 -18289.229,E2 -18289.229} C_VEL
LIN {X 0,Y 273.792,Z 859.808,A -85,B 0,C 180,E1 -18291.058,E2 -18291.058} C_VEL
LIN {X 0,Y 274.76,Z 853.861,A -85,B 0,C 180,E1 -18291.995,E2 -18291.995} C_VEL
LIN {X 0,Y 273.779,Z 848.952,A -85,B 0,C 180,E1 -18292.87,E2 -18292.87} C_VEL
LIN {X 0,Y 270.598,Z 838.477,A -85,B 0,C 180,E1 -18294.628,E2 -18294.628} C_VEL
LIN {X 0,Y 266.458,Z 827.594,A -85,B 0,C 180,E1 -18296.263,E2 -18296.263} C_VEL
LIN {X 0,Y 263.266,Z 819.692,A -85,B 0,C 180,E1 -18297.317,E2 -18297.317} C_VEL
LIN {X 0,Y 263.128,Z 819.711,A -85,B 0,C 180,E1 -18302.285,E2 -18302.285} C_VEL
LIN {X 0,Y 263.183,Z 819.704,A -85,B 0,C 180,E1 -18305.975,E2 -18305.975} C_VEL
LIN {X 0,Y 263.155,Z 819.706,A -85,B 0,C 180,E1 -18309.859,E2 -18309.859} C_VEL
LIN {X 0,Y 263.183,Z 819.703,A -85,B 0,C 180,E1 -18313.862,E2 -18313.862} C_VEL
LIN {X 0,Y 263.205,Z 819.696,A -85,B 0,C 180,E1 -18318.382,E2 -18318.382} C_VEL
LIN {X 0,Y 263.178,Z 819.696,A -85,B 0,C 180,E1 -18322.106,E2 -18322.106} C_VEL
LIN {X 0,Y 263.172,Z 819.694,A -85,B 0,C 180,E1 -18325.888,E2 -18325.888} C_VEL
LIN {X 0,Y 263.138,Z 819.7,A -85,B 0,C 180,E1 -18329.505,E2 -18329.505} C_VEL
LIN {X 0,Y 263.18,Z 819.7,A -85,B 0,C 180,E1 -18333.001,E2 -18333.001} C_VEL
LIN {X 0,Y 263.17,Z 819.702,A -85,B 0,C 180,E1 -18336.386,E2 -18336.386} C_VEL
LIN {X 0,Y 263.249,Z 819.688,A -85,B 0,C 180,E1 -18339.692,E2 -18339.692} C_VEL
LIN {X 0,Y 263.336,Z 819.672,A -85,B 0,C 180,E1 -18344.521,E2 -18344.521} C_VEL
LIN {X 0,Y 263.359,Z 819.678,A -85,B 0,C 180,E1 -18349.234,E2 -18349.234} C_VEL
LIN {X 0,Y 263.554,Z 819.655,A -85,B 0,C 180,E1 -18352.338,E2 -18352.338} C_VEL
LIN {X 0,Y 263.736,Z 819.634,A -85,B 0,C 180,E1 -18358.473,E2 -18358.473} C_VEL
LIN {X 0,Y 263.735,Z 819.637,A -85,B 0,C 180,E1 -18361.527,E2 -18361.527} C_VEL
LIN {X 0,Y 263.547,Z 819.66,A -85,B 0,C 180,E1 -18367.662,E2 -18367.662} C_VEL
LIN {X 0,Y 263.359,Z 819.678,A -85,B 0,C 180,E1 -18370.766,E2 -18370.766} C_VEL
LIN {X 0,Y 263.336,Z 819.684,A -85,B 0,C 180,E1 -18375.479,E2 -18375.479} C_VEL
LIN {X 0,Y 263.247,Z 819.697,A -85,B 0,C 180,E1 -18380.308,E2 -18380.308} C_VEL
LIN {X 0,Y 263.118,Z 819.71,A -85,B 0,C 180,E1 -18382.106,E2 -18382.106} C_VEL
LIN {X 0,Y 262.422,Z 819.797,A -85,B 0,C 180,E1 -18383.383,E2 -18383.383} C_VEL
LIN {X 0,Y 259.596,Z 820.148,A -85,B 0,C 180,E1 -18385.466,E2 -18385.466} C_VEL
LIN {X 0,Y 257.203,Z 820.448,A -85,B 0,C 180,E1 -18387.16,E2 -18387.16} C_VEL
LIN {X 0,Y 256.154,Z 820.577,A -85,B 0,C 180,E1 -18388.472,E2 -18388.472} C_VEL
LIN {X 0,Y 256.055,Z 820.588,A -85,B 0,C 180,E1 -18388.916,E2 -18388.916} C_VEL
LIN {X 0,Y 256.053,Z 820.589,A -85,B 0,C 180,E1 -18393.295,E2 -18393.295} C_VEL
LIN {X 0,Y 256.146,Z 820.804,A -85,B 0,C 180,E1 -18394.813,E2 -18394.813} C_VEL
LIN {X 0,Y 257.424,Z 826.973,A -85,B 0,C 180,E1 -18398.898,E2 -18398.898} C_VEL
LIN {X 0,Y 258.732,Z 833.392,A -85,B 0,C 180,E1 -18402.832,E2 -18402.832} C_VEL
LIN {X 0,Y 260.129,Z 840.434,A -85,B 0,C 180,E1 -18406.842,E2 -18406.842} C_VEL
LIN {X 0,Y 261.32,Z 847.487,A -85,B 0,C 180,E1 -18410.62,E2 -18410.62} C_VEL
LIN {X 0,Y 261.117,Z 849.776,A -85,B 0,C 180,E1 -18411.758,E2 -18411.758} C_VEL
LIN {X 0,Y 259.553,Z 857.304,A -85,B 0,C 180,E1 -18415.35,E2 -18415.35} C_VEL
LIN {X 0,Y 257.595,Z 868.29,A -85,B 0,C 180,E1 -18420.591,E2 -18420.591} C_VEL
LIN {X 0,Y 257.434,Z 869.369,A -85,B 0,C 180,E1 -18421.113,E2 -18421.113} C_VEL
LIN {X 0,Y 259.814,Z 883.609,A -85,B 0,C 180,E1 -18422.074,E2 -18422.074} C_VEL
LIN {X 0,Y 261.285,Z 896.122,A -85,B 0,C 180,E1 -18423.151,E2 -18423.151} C_VEL
LIN {X 0,Y 261.945,Z 908.409,A -85,B 0,C 180,E1 -18424.443,E2 -18424.443} C_VEL
LIN {X 0,Y 261.969,Z 919.737,A -85,B 0,C 180,E1 -18425.884,E2 -18425.884} C_VEL
LIN {X 0,Y 261.343,Z 931.434,A -85,B 0,C 180,E1 -18427.679,E2 -18427.679} C_VEL
LIN {X 0,Y 260.61,Z 941.05,A -85,B 0,C 180,E1 -18429.481,E2 -18429.481} C_VEL
LIN {X 0,Y 258.802,Z 949.684,A -85,B 0,C 180,E1 -18431.396,E2 -18431.396} C_VEL
LIN {X 0,Y 257.056,Z 957.734,A -85,B 0,C 180,E1 -18433.6,E2 -18433.6} C_VEL
LIN {X 0,Y 255.994,Z 965.045,A -85,B 0,C 180,E1 -18436.104,E2 -18436.104} C_VEL
LIN {X 0,Y 255.24,Z 971.408,A -85,B 0,C 180,E1 -18438.89,E2 -18438.89} C_VEL
LIN {X 0,Y 255.035,Z 975.595,A -85,B 0,C 180,E1 -18441.285,E2 -18441.285} C_VEL
LIN {X 0,Y 255.147,Z 978.73,A -85,B 0,C 180,E1 -18443.677,E2 -18443.677} C_VEL
LIN {X 0,Y 255.397,Z 980.251,A -85,B 0,C 180,E1 -18445.268,E2 -18445.268} C_VEL
LIN {X 0,Y 255.594,Z 981.337,A -85,B 0,C 180,E1 -18446.85,E2 -18446.85} C_VEL
LIN {X 0,Y 255.771,Z 982.006,A -85,B 0,C 180,E1 -18448.428,E2 -18448.428} C_VEL
LIN {X 0,Y 255.937,Z 982.255,A -85,B 0,C 180,E1 -18450.003,E2 -18450.003} C_VEL
LIN {X 0,Y 255.772,Z 981.996,A -85,B 0,C 180,E1 -18451.577,E2 -18451.577} C_VEL
LIN {X 0,Y 255.602,Z 981.32,A -85,B 0,C 180,E1 -18453.155,E2 -18453.155} C_VEL
LIN {X 0,Y 255.421,Z 980.229,A -85,B 0,C 180,E1 -18454.738,E2 -18454.738} C_VEL
LIN {X 0,Y 255.143,Z 977.392,A -85,B 0,C 180,E1 -18457.416,E2 -18457.416} C_VEL
LIN {X 0,Y 255.514,Z 970.091,A -85,B 0,C 180,E1 -18462.714,E2 -18462.714} C_VEL
LIN {X 0,Y 257.002,Z 964.196,A -85,B 0,C 180,E1 -18465.873,E2 -18465.873} C_VEL
LIN {X 0,Y 259.007,Z 957.575,A -85,B 0,C 180,E1 -18468.594,E2 -18468.594} C_VEL
LIN {X 0,Y 261.398,Z 950.812,A -85,B 0,C 180,E1 -18470.872,E2 -18470.872} C_VEL
LIN {X 0,Y 263.664,Z 944.346,A -85,B 0,C 180,E1 -18472.739,E2 -18472.739} C_VEL
LIN {X 0,Y 266.45,Z 933.917,A -85,B 0,C 180,E1 -18475.382,E2 -18475.382} C_VEL
LIN {X 0,Y 269.484,Z 922.98,A -85,B 0,C 180,E1 -18477.665,E2 -18477.665} C_VEL
LIN {X 0,Y 271.143,Z 913.823,A -85,B 0,C 180,E1 -18479.506,E2 -18479.506} C_VEL
LIN {X 0,Y 272.388,Z 903.099,A -85,B 0,C 180,E1 -18481.63,E2 -18481.63} C_VEL
LIN {X 0,Y 273.077,Z 892.581,A -85,B 0,C 180,E1 -18483.754,E2 -18483.754} C_VEL
LIN {X 0,Y 273.391,Z 882.686,A -85,B 0,C 180,E1 -18485.883,E2 -18485.883} C_VEL
LIN {X 0,Y 273.512,Z 876.733,A -85,B 0,C 180,E1 -18487.197,E2 -18487.197} C_VEL
LIN {X 0,Y 273.689,Z 868.603,A -85,B 0,C 180,E1 -18489.22,E2 -18489.22} C_VEL
LIN {X 0,Y 273.55,Z 862.752,A -85,B 0,C 180,E1 -18491.009,E2 -18491.009} C_VEL
LIN {X 0,Y 273.361,Z 857.88,A -85,B 0,C 180,E1 -18493.051,E2 -18493.051} C_VEL
LIN {X 0,Y 273.313,Z 854.537,A -85,B 0,C 180,E1 -18495.099,E2 -18495.099} C_VEL
LIN {X 0,Y 273.422,Z 853.322,A -85,B 0,C 180,E1 -18496.052,E2 -18496.052} C_VEL
LIN {X 0,Y 273.958,Z 851.413,A -85,B 0,C 180,E1 -18498.164,E2 -18498.164} C_VEL
LIN {X 0,Y 274.866,Z 850.66,A -85,B 0,C 180,E1 -18500.266,E2 -18500.266} C_VEL
LIN {X 0,Y 276.148,Z 851.055,A -85,B 0,C 180,E1 -18502.352,E2 -18502.352} C_VEL
LIN {X 0,Y 278.199,Z 853.367,A -85,B 0,C 180,E1 -18505.256,E2 -18505.256} C_VEL
LIN {X 0,Y 279.793,Z 855.989,A -85,B 0,C 180,E1 -18507.149,E2 -18507.149} C_VEL
LIN {X 0,Y 281.418,Z 862.312,A -85,B 0,C 180,E1 -18510.035,E2 -18510.035} C_VEL
LIN {X 0,Y 282.37,Z 868.644,A -85,B 0,C 180,E1 -18512.465,E2 -18512.465} C_VEL
LIN {X 0,Y 282.568,Z 871.687,A -85,B 0,C 180,E1 -18513.562,E2 -18513.562} C_VEL
LIN {X 0,Y 282.424,Z 873.347,A -85,B 0,C 180,E1 -18514.045,E2 -18514.045} C_VEL
LIN {X 0,Y 278.398,Z 882.638,A -85,B 0,C 180,E1 -18516.177,E2 -18516.177} C_VEL
LIN {X 0,Y 274.795,Z 889.774,A -85,B 0,C 180,E1 -18518.232,E2 -18518.232} C_VEL
LIN {X 0,Y 271.515,Z 895.665,A -85,B 0,C 180,E1 -18520.336,E2 -18520.336} C_VEL
LIN {X 0,Y 268.676,Z 900.36,A -85,B 0,C 180,E1 -18522.493,E2 -18522.493} C_VEL
LIN {X 0,Y 266.04,Z 904.137,A -85,B 0,C 180,E1 -18524.682,E2 -18524.682} C_VEL
LIN {X 0,Y 263.062,Z 907.563,A -85,B 0,C 180,E1 -18527.659,E2 -18527.659} C_VEL
LIN {X 0,Y 260.501,Z 909.339,A -85,B 0,C 180,E1 -18530.684,E2 -18530.684} C_VEL
LIN {X 0,Y 259.669,Z 909.662,A -85,B 0,C 180,E1 -18532.223,E2 -18532.223} C_VEL
LIN {X 0,Y 258.853,Z 909.603,A -85,B 0,C 180,E1 -18533.765,E2 -18533.765} C_VEL
LIN {X 0,Y 257.626,Z 908.23,A -85,B 0,C 180,E1 -18536.872,E2 -18536.872} C_VEL
LIN {X 0,Y 256.635,Z 905.3,A -85,B 0,C 180,E1 -18540,E2 -18540} C_VEL
LIN {X 0,Y 256.477,Z 901.976,A -85,B 0,C 180,E1 -18542.356,E2 -18542.356} C_VEL
LIN {X 0,Y 256.232,Z 897.649,A -85,B 0,C 180,E1 -18544.72,E2 -18544.72} C_VEL
LIN {X 0,Y 256.728,Z 892.175,A -85,B 0,C 180,E1 -18547.076,E2 -18547.076} C_VEL
LIN {X 0,Y 257.148,Z 885.451,A -85,B 0,C 180,E1 -18549.438,E2 -18549.438} C_VEL
LIN {X 0,Y 257.809,Z 877.381,A -85,B 0,C 180,E1 -18551.798,E2 -18551.798} C_VEL
LIN {X 0,Y 258.723,Z 867.35,A -85,B 0,C 180,E1 -18554.151,E2 -18554.151} C_VEL
LIN {X 0,Y 259.688,Z 856.104,A -85,B 0,C 180,E1 -18556.307,E2 -18556.307} C_VEL
LIN {X 0,Y 260.777,Z 844.958,A -85,B 0,C 180,E1 -18558.055,E2 -18558.055} C_VEL
LIN {X 0,Y 261,Z 840.889,A -85,B 0,C 180,E1 -18558.612,E2 -18558.612} C_VEL
LIN {X 0,Y 258.017,Z 828.567,A -85,B 0,C 180,E1 -18560.227,E2 -18560.227} C_VEL
LIN {X 0,Y 256.135,Z 820.567,A -85,B 0,C 180,E1 -18561.145,E2 -18561.145} C_VEL
LIN {X 0,Y 256.09,Z 820.583,A -85,B 0,C 180,E1 -18565.086,E2 -18565.086} C_VEL
LIN {X 0,Y 256.084,Z 820.579,A -85,B 0,C 180,E1 -18568.568,E2 -18568.568} C_VEL
LIN {X 0,Y 256.077,Z 820.577,A -85,B 0,C 180,E1 -18571.698,E2 -18571.698} C_VEL
LIN {X 0,Y 256.087,Z 820.582,A -85,B 0,C 180,E1 -18575.192,E2 -18575.192} C_VEL
LIN {X 0,Y 256.072,Z 820.582,A -85,B 0,C 180,E1 -18579.142,E2 -18579.142} C_VEL
LIN {X 0,Y 256.03,Z 820.588,A -85,B 0,C 180,E1 -18583.334,E2 -18583.334} C_VEL
LIN {X 0,Y 256.038,Z 820.591,A -85,B 0,C 180,E1 -18587.828,E2 -18587.828} C_VEL
LIN {X 0,Y 256.123,Z 820.576,A -85,B 0,C 180,E1 -18592.727,E2 -18592.727} C_VEL
LIN {X 0,Y 256.075,Z 820.585,A -85,B 0,C 180,E1 -18596.706,E2 -18596.706} C_VEL
LIN {X 0,Y 256.111,Z 820.575,A -85,B 0,C 180,E1 -18600.397,E2 -18600.397} C_VEL
LIN {X 0,Y 256.197,Z 820.566,A -85,B 0,C 180,E1 -18601.992,E2 -18601.992} C_VEL
LIN {X 0,Y 257.078,Z 823.147,A -85,B 0,C 180,E1 -18602.304,E2 -18602.304} C_VEL
LIN {X 0,Y 261.213,Z 832.693,A -85,B 0,C 180,E1 -18603.715,E2 -18603.715} C_VEL
LIN {X 0,Y 264.838,Z 842.803,A -85,B 0,C 180,E1 -18605.353,E2 -18605.353} C_VEL
LIN {X 0,Y 267.644,Z 852.984,A -85,B 0,C 180,E1 -18607.186,E2 -18607.186} C_VEL
LIN {X 0,Y 268.143,Z 855.236,A -85,B 0,C 180,E1 -18607.614,E2 -18607.614} C_VEL
LIN {X 0,Y 266.547,Z 864.352,A -85,B 0,C 180,E1 -18609.146,E2 -18609.146} C_VEL
LIN {X 0,Y 264.854,Z 873.372,A -85,B 0,C 180,E1 -18611.028,E2 -18611.028} C_VEL
LIN {X 0,Y 262.79,Z 882.152,A -85,B 0,C 180,E1 -18613.289,E2 -18613.289} C_VEL
LIN {X 0,Y 261.316,Z 888.958,A -85,B 0,C 180,E1 -18615.515,E2 -18615.515} C_VEL
LIN {X 0,Y 260.247,Z 893.886,A -85,B 0,C 180,E1 -18617.521,E2 -18617.521} C_VEL
LIN {X 0,Y 258.821,Z 898.523,A -85,B 0,C 180,E1 -18619.831,E2 -18619.831} C_VEL
LIN {X 0,Y 257.837,Z 902.045,A -85,B 0,C 180,E1 -18622.164,E2 -18622.164} C_VEL
LIN {X 0,Y 257.357,Z 903.86,A -85,B 0,C 180,E1 -18623.726,E2 -18623.726} C_VEL
LIN {X 0,Y 257.24,Z 905.189,A -85,B 0,C 180,E1 -18625.296,E2 -18625.296} C_VEL
LIN {X 0,Y 256.756,Z 906.767,A -85,B 0,C 180,E1 -18628.429,E2 -18628.429} C_VEL
LIN {X 0,Y 256.688,Z 906.996,A -85,B 0,C 180,E1 -18629.997,E2 -18629.997} C_VEL
LIN {X 0,Y 256.968,Z 906.225,A -85,B 0,C 180,E1 -18633.133,E2 -18633.133} C_VEL
LIN {X 0,Y 257.226,Z 905.281,A -85,B 0,C 180,E1 -18634.699,E2 -18634.699} C_VEL
LIN {X 0,Y 257.343,Z 903.992,A -85,B 0,C 180,E1 -18636.269,E2 -18636.269} C_VEL
LIN {X 0,Y 258.101,Z 901.184,A -85,B 0,C 180,E1 -18638.61,E2 -18638.61} C_VEL
LIN {X 0,Y 259.345,Z 897.338,A -85,B 0,C 180,E1 -18640.932,E2 -18640.932} C_VEL
LIN {X 0,Y 260.597,Z 892.423,A -85,B 0,C 180,E1 -18643.249,E2 -18643.249} C_VEL
LIN {X 0,Y 261.935,Z 886.247,A -85,B 0,C 180,E1 -18645.561,E2 -18645.561} C_VEL
LIN {X 0,Y 263.742,Z 878.471,A -85,B 0,C 180,E1 -18647.842,E2 -18647.842} C_VEL
LIN {X 0,Y 265.425,Z 870.534,A -85,B 0,C 180,E1 -18649.727,E2 -18649.727} C_VEL
LIN {X 0,Y 267.258,Z 860.835,A -85,B 0,C 180,E1 -18651.599,E2 -18651.599} C_VEL
LIN {X 0,Y 268.166,Z 854.903,A -85,B 0,C 180,E1 -18652.565,E2 -18652.565} C_VEL
LIN {X 0,Y 265.839,Z 845.992,A -85,B 0,C 180,E1 -18654.219,E2 -18654.219} C_VEL
LIN {X 0,Y 262.543,Z 836.108,A -85,B 0,C 180,E1 -18655.871,E2 -18655.871} C_VEL
LIN {X 0,Y 257.838,Z 824.618,A -85,B 0,C 180,E1 -18657.602,E2 -18657.602} C_VEL
LIN {X 0,Y 256.287,Z 821.216,A -85,B 0,C 180,E1 -18658.077,E2 -18658.077} C_VEL
LIN {X 0,Y 256.154,Z 820.578,A -85,B 0,C 180,E1 -18658.188,E2 -18658.188} C_VEL
LIN {X 0,Y 256.077,Z 820.589,A -85,B 0,C 180,E1 -18661.702,E2 -18661.702} C_VEL
LIN {X 0,Y 256.115,Z 820.583,A -85,B 0,C 180,E1 -18665.184,E2 -18665.184} C_VEL
LIN {X 0,Y 256.102,Z 820.584,A -85,B 0,C 180,E1 -18669.132,E2 -18669.132} C_VEL
LIN {X 0,Y 256.134,Z 820.579,A -85,B 0,C 180,E1 -18673.307,E2 -18673.307} C_VEL
LIN {X 0,Y 256.153,Z 820.57,A -85,B 0,C 180,E1 -18677.794,E2 -18677.794} C_VEL
LIN {X 0,Y 256.138,Z 820.573,A -85,B 0,C 180,E1 -18680.87,E2 -18680.87} C_VEL
LIN {X 0,Y 256.11,Z 820.577,A -85,B 0,C 180,E1 -18684.811,E2 -18684.811} C_VEL
LIN {X 0,Y 256.08,Z 820.585,A -85,B 0,C 180,E1 -18688.57,E2 -18688.57} C_VEL
LIN {X 0,Y 256.129,Z 820.579,A -85,B 0,C 180,E1 -18692.194,E2 -18692.194} C_VEL
LIN {X 0,Y 256.154,Z 820.575,A -85,B 0,C 180,E1 -18695.698,E2 -18695.698} C_VEL
LIN {X 0,Y 256.153,Z 820.571,A -85,B 0,C 180,E1 -18699.104,E2 -18699.104} C_VEL
LIN {X 0,Y 256.285,Z 820.552,A -85,B 0,C 180,E1 -18704.084,E2 -18704.084} C_VEL
LIN {X 0,Y 256.295,Z 820.561,A -85,B 0,C 180,E1 -18708.933,E2 -18708.933} C_VEL
LIN {X 0,Y 256.522,Z 820.531,A -85,B 0,C 180,E1 -18712.126,E2 -18712.126} C_VEL
LIN {X 0,Y 256.699,Z 820.511,A -85,B 0,C 180,E1 -18718.431,E2 -18718.431} C_VEL
LIN {X 0,Y 256.698,Z 820.514,A -85,B 0,C 180,E1 -18721.569,E2 -18721.569} C_VEL
LIN {X 0,Y 256.517,Z 820.534,A -85,B 0,C 180,E1 -18727.874,E2 -18727.874} C_VEL
LIN {X 0,Y 256.295,Z 820.559,A -85,B 0,C 180,E1 -18731.067,E2 -18731.067} C_VEL
LIN {X 0,Y 256.285,Z 820.562,A -85,B 0,C 180,E1 -18735.916,E2 -18735.916} C_VEL
LIN {X 0,Y 256.146,Z 820.58,A -85,B 0,C 180,E1 -18740.897,E2 -18740.897} C_VEL
LIN {X 0,Y 256.118,Z 820.581,A -85,B 0,C 180,E1 -18745.113,E2 -18745.113} C_VEL
LIN {X 0,Y 256.055,Z 820.588,A -85,B 0,C 180,E1 -18748.916,E2 -18748.916} C_VEL
LIN {X 0,Y 255.363,Z 820.675,A -85,B 0,C 180,E1 -18749.791,E2 -18749.791} C_VEL
LIN {X 0,Y 252.549,Z 821.026,A -85,B 0,C 180,E1 -18751.165,E2 -18751.165} C_VEL
LIN {X 0,Y 249.715,Z 821.377,A -85,B 0,C 180,E1 -18752.568,E2 -18752.568} C_VEL
LIN {X 0,Y 249.024,Z 821.465,A -85,B 0,C 180,E1 -18753.475,E2 -18753.475} C_VEL
LIN {X 0,Y 249.039,Z 821.534,A -85,B 0,C 180,E1 -18753.873,E2 -18753.873} C_VEL
LIN {X 0,Y 250.079,Z 826.248,A -85,B 0,C 180,E1 -18757.173,E2 -18757.173} C_VEL
LIN {X 0,Y 251.274,Z 832.08,A -85,B 0,C 180,E1 -18760.965,E2 -18760.965} C_VEL
LIN {X 0,Y 252.596,Z 838.861,A -85,B 0,C 180,E1 -18765.062,E2 -18765.062} C_VEL
LIN {X 0,Y 253.71,Z 844.751,A -85,B 0,C 180,E1 -18768.411,E2 -18768.411} C_VEL
LIN {X 0,Y 254.317,Z 848.968,A -85,B 0,C 180,E1 -18770.694,E2 -18770.694} C_VEL
LIN {X 0,Y 253.396,Z 853.779,A -85,B 0,C 180,E1 -18773.096,E2 -18773.096} C_VEL
LIN {X 0,Y 251.608,Z 862.482,A -85,B 0,C 180,E1 -18777.391,E2 -18777.391} C_VEL
LIN {X 0,Y 250.613,Z 868.265,A -85,B 0,C 180,E1 -18780.248,E2 -18780.248} C_VEL
LIN {X 0,Y 253.101,Z 882.765,A -85,B 0,C 180,E1 -18781.281,E2 -18781.281} C_VEL
LIN {X 0,Y 254.584,Z 895.727,A -85,B 0,C 180,E1 -18782.451,E2 -18782.451} C_VEL
LIN {X 0,Y 255.255,Z 908.513,A -85,B 0,C 180,E1 -18783.866,E2 -18783.866} C_VEL
LIN {X 0,Y 255.228,Z 919.481,A -85,B 0,C 180,E1 -18785.326,E2 -18785.326} C_VEL
LIN {X 0,Y 254.563,Z 930.359,A -85,B 0,C 180,E1 -18787.051,E2 -18787.051} C_VEL
LIN {X 0,Y 253.809,Z 939.985,A -85,B 0,C 180,E1 -18788.905,E2 -18788.905} C_VEL
LIN {X 0,Y 252.013,Z 948.632,A -85,B 0,C 180,E1 -18790.875,E2 -18790.875} C_VEL
LIN {X 0,Y 250.1,Z 957.027,A -85,B 0,C 180,E1 -18793.245,E2 -18793.245} C_VEL
LIN {X 0,Y 249.025,Z 963.992,A -85,B 0,C 180,E1 -18795.706,E2 -18795.706} C_VEL
LIN {X 0,Y 248.198,Z 970.355,A -85,B 0,C 180,E1 -18798.571,E2 -18798.571} C_VEL
LIN {X 0,Y 247.991,Z 974.549,A -85,B 0,C 180,E1 -18801.036,E2 -18801.036} C_VEL
LIN {X 0,Y 248.079,Z 977.687,A -85,B 0,C 180,E1 -18803.496,E2 -18803.496} C_VEL
LIN {X 0,Y 248.325,Z 979.209,A -85,B 0,C 180,E1 -18805.132,E2 -18805.132} C_VEL
LIN {X 0,Y 248.535,Z 980.299,A -85,B 0,C 180,E1 -18806.761,E2 -18806.761} C_VEL
LIN {X 0,Y 248.728,Z 980.972,A -85,B 0,C 180,E1 -18808.384,E2 -18808.384} C_VEL
LIN {X 0,Y 248.907,Z 981.223,A -85,B 0,C 180,E1 -18810.003,E2 -18810.003} C_VEL
LIN {X 0,Y 248.729,Z 980.962,A -85,B 0,C 180,E1 -18811.622,E2 -18811.622} C_VEL
LIN {X 0,Y 248.544,Z 980.282,A -85,B 0,C 180,E1 -18813.245,E2 -18813.245} C_VEL
LIN {X 0,Y 248.349,Z 979.187,A -85,B 0,C 180,E1 -18814.873,E2 -18814.873} C_VEL
LIN {X 0,Y 248.08,Z 976.545,A -85,B 0,C 180,E1 -18817.459,E2 -18817.459} C_VEL
LIN {X 0,Y 248.031,Z 973.448,A -85,B 0,C 180,E1 -18819.791,E2 -18819.791} C_VEL
LIN {X 0,Y 248.316,Z 970.507,A -85,B 0,C 180,E1 -18822.258,E2 -18822.258} C_VEL
LIN {X 0,Y 249.198,Z 966.751,A -85,B 0,C 180,E1 -18824.707,E2 -18824.707} C_VEL
LIN {X 0,Y 250.662,Z 962.15,A -85,B 0,C 180,E1 -18827.124,E2 -18827.124} C_VEL
LIN {X 0,Y 253.023,Z 955.441,A -85,B 0,C 180,E1 -18829.895,E2 -18829.895} C_VEL
LIN {X 0,Y 255.732,Z 948.634,A -85,B 0,C 180,E1 -18832.205,E2 -18832.205} C_VEL
LIN {X 0,Y 257.834,Z 942.193,A -85,B 0,C 180,E1 -18834.136,E2 -18834.136} C_VEL
LIN {X 0,Y 261.191,Z 931.827,A -85,B 0,C 180,E1 -18836.791,E2 -18836.791} C_VEL
LIN {X 0,Y 264.193,Z 921.474,A -85,B 0,C 180,E1 -18839.047,E2 -18839.047} C_VEL
LIN {X 0,Y 266.113,Z 911.34,A -85,B 0,C 180,E1 -18841.222,E2 -18841.222} C_VEL
LIN {X 0,Y 267.56,Z 900.732,A -85,B 0,C 180,E1 -18843.48,E2 -18843.48} C_VEL
LIN {X 0,Y 268.527,Z 889.925,A -85,B 0,C 180,E1 -18845.893,E2 -18845.893} C_VEL
LIN {X 0,Y 269.325,Z 880.273,A -85,B 0,C 180,E1 -18848.196,E2 -18848.196} C_VEL
LIN {X 0,Y 269.816,Z 872.5,A -85,B 0,C 180,E1 -18850.258,E2 -18850.258} C_VEL
LIN {X 0,Y 270.122,Z 867.759,A -85,B 0,C 180,E1 -18851.798,E2 -18851.798} C_VEL
LIN {X 0,Y 270.232,Z 864.341,A -85,B 0,C 180,E1 -18853.264,E2 -18853.264} C_VEL
LIN {X 0,Y 270.345,Z 860.792,A -85,B 0,C 180,E1 -18855.42,E2 -18855.42} C_VEL
LIN {X 0,Y 270.769,Z 858.512,A -85,B 0,C 180,E1 -18857.558,E2 -18857.558} C_VEL
LIN {X 0,Y 271.514,Z 857.289,A -85,B 0,C 180,E1 -18859.676,E2 -18859.676} C_VEL
LIN {X 0,Y 272.503,Z 857.204,A -85,B 0,C 180,E1 -18861.759,E2 -18861.759} C_VEL
LIN {X 0,Y 273.687,Z 858.315,A -85,B 0,C 180,E1 -18863.799,E2 -18863.799} C_VEL
LIN {X 0,Y 274.999,Z 860.167,A -85,B 0,C 180,E1 -18865.789,E2 -18865.789} C_VEL
LIN {X 0,Y 275.83,Z 862.321,A -85,B 0,C 180,E1 -18867.231,E2 -18867.231} C_VEL
LIN {X 0,Y 276.763,Z 867.398,A -85,B 0,C 180,E1 -18869.702,E2 -18869.702} C_VEL
LIN {X 0,Y 277.198,Z 872.127,A -85,B 0,C 180,E1 -18871.67,E2 -18871.67} C_VEL
LIN {X 0,Y 277.21,Z 876.257,A -85,B 0,C 180,E1 -18873.207,E2 -18873.207} C_VEL
LIN {X 0,Y 272.524,Z 886.122,A -85,B 0,C 180,E1 -18875.631,E2 -18875.631} C_VEL
LIN {X 0,Y 268.152,Z 893.886,A -85,B 0,C 180,E1 -18878.07,E2 -18878.07} C_VEL
LIN {X 0,Y 264.267,Z 899.997,A -85,B 0,C 180,E1 -18880.584,E2 -18880.584} C_VEL
LIN {X 0,Y 260.418,Z 905.243,A -85,B 0,C 180,E1 -18883.539,E2 -18883.539} C_VEL
LIN {X 0,Y 257.848,Z 907.939,A -85,B 0,C 180,E1 -18885.8,E2 -18885.8} C_VEL
LIN {X 0,Y 256.36,Z 909.347,A -85,B 0,C 180,E1 -18887.331,E2 -18887.331} C_VEL
LIN {X 0,Y 254.985,Z 910.288,A -85,B 0,C 180,E1 -18888.876,E2 -18888.876} C_VEL
LIN {X 0,Y 252.788,Z 911.07,A -85,B 0,C 180,E1 -18892.009,E2 -18892.009} C_VEL
LIN {X 0,Y 251.237,Z 910.228,A -85,B 0,C 180,E1 -18895.186,E2 -18895.186} C_VEL
LIN {X 0,Y 250.629,Z 909.248,A -85,B 0,C 180,E1 -18896.785,E2 -18896.785} C_VEL
LIN {X 0,Y 249.586,Z 905.986,A -85,B 0,C 180,E1 -18900,E2 -18900} C_VEL
LIN {X 0,Y 249.403,Z 902.465,A -85,B 0,C 180,E1 -18902.423,E2 -18902.423} C_VEL
LIN {X 0,Y 249.17,Z 897.935,A -85,B 0,C 180,E1 -18904.854,E2 -18904.854} C_VEL
LIN {X 0,Y 249.677,Z 892.255,A -85,B 0,C 180,E1 -18907.277,E2 -18907.277} C_VEL
LIN {X 0,Y 250.05,Z 886.578,A -85,B 0,C 180,E1 -18909.301,E2 -18909.301} C_VEL
LIN {X 0,Y 250.682,Z 878.497,A -85,B 0,C 180,E1 -18911.728,E2 -18911.728} C_VEL
LIN {X 0,Y 251.615,Z 868.466,A -85,B 0,C 180,E1 -18914.147,E2 -18914.147} C_VEL
LIN {X 0,Y 252.577,Z 857.237,A -85,B 0,C 180,E1 -18916.364,E2 -18916.364} C_VEL
LIN {X 0,Y 253.765,Z 845.374,A -85,B 0,C 180,E1 -18918.27,E2 -18918.27} C_VEL
LIN {X 0,Y 253.927,Z 841.563,A -85,B 0,C 180,E1 -18918.803,E2 -18918.803} C_VEL
LIN {X 0,Y 250.826,Z 828.757,A -85,B 0,C 180,E1 -18920.502,E2 -18920.502} C_VEL
LIN {X 0,Y 249.067,Z 821.447,A -85,B 0,C 180,E1 -18921.376,E2 -18921.376} C_VEL
LIN {X 0,Y 249.051,Z 821.459,A -85,B 0,C 180,E1 -18925.438,E2 -18925.438} C_VEL
LIN {X 0,Y 249.032,Z 821.458,A -85,B 0,C 180,E1 -18928.967,E2 -18928.967} C_VEL
LIN {X 0,Y 249.034,Z 821.449,A -85,B 0,C 180,E1 -18932.426,E2 -18932.426} C_VEL
LIN {X 0,Y 249.021,Z 821.459,A -85,B 0,C 180,E1 -18936.347,E2 -18936.347} C_VEL
LIN {X 0,Y 248.986,Z 821.467,A -85,B 0,C 180,E1 -18940.482,E2 -18940.482} C_VEL
LIN {X 0,Y 248.97,Z 821.471,A -85,B 0,C 180,E1 -18944.887,E2 -18944.887} C_VEL
LIN {X 0,Y 248.985,Z 821.468,A -85,B 0,C 180,E1 -18947.353,E2 -18947.353} C_VEL
LIN {X 0,Y 249.046,Z 821.461,A -85,B 0,C 180,E1 -18952.2,E2 -18952.2} C_VEL
LIN {X 0,Y 249.05,Z 821.461,A -85,B 0,C 180,E1 -18955.638,E2 -18955.638} C_VEL
LIN {X 0,Y 249.055,Z 821.456,A -85,B 0,C 180,E1 -18959.471,E2 -18959.471} C_VEL
LIN {X 0,Y 249.105,Z 821.539,A -85,B 0,C 180,E1 -18961.106,E2 -18961.106} C_VEL
LIN {X 0,Y 250.134,Z 824.314,A -85,B 0,C 180,E1 -18961.465,E2 -18961.465} C_VEL
LIN {X 0,Y 254.601,Z 834.393,A -85,B 0,C 180,E1 -18963.045,E2 -18963.045} C_VEL
LIN {X 0,Y 258.266,Z 844.69,A -85,B 0,C 180,E1 -18964.798,E2 -18964.798} C_VEL
LIN {X 0,Y 260.959,Z 854.375,A -85,B 0,C 180,E1 -18966.621,E2 -18966.621} C_VEL
LIN {X 0,Y 261.563,Z 856.905,A -85,B 0,C 180,E1 -18967.127,E2 -18967.127} C_VEL
LIN {X 0,Y 259.576,Z 867.32,A -85,B 0,C 180,E1 -18968.974,E2 -18968.974} C_VEL
LIN {X 0,Y 257.863,Z 875.999,A -85,B 0,C 180,E1 -18970.907,E2 -18970.907} C_VEL
LIN {X 0,Y 256.071,Z 883.186,A -85,B 0,C 180,E1 -18972.837,E2 -18972.837} C_VEL
LIN {X 0,Y 254.567,Z 889.867,A -85,B 0,C 180,E1 -18975.077,E2 -18975.077} C_VEL
LIN {X 0,Y 253.395,Z 894.919,A -85,B 0,C 180,E1 -18977.178,E2 -18977.178} C_VEL
LIN {X 0,Y 251.91,Z 899.556,A -85,B 0,C 180,E1 -18979.549,E2 -18979.549} C_VEL
LIN {X 0,Y 250.879,Z 903.078,A -85,B 0,C 180,E1 -18981.945,E2 -18981.945} C_VEL
LIN {X 0,Y 250.403,Z 904.888,A -85,B 0,C 180,E1 -18983.551,E2 -18983.551} C_VEL
LIN {X 0,Y 250.24,Z 906.22,A -85,B 0,C 180,E1 -18985.164,E2 -18985.164} C_VEL
LIN {X 0,Y 249.735,Z 907.798,A -85,B 0,C 180,E1 -18988.385,E2 -18988.385} C_VEL
LIN {X 0,Y 249.664,Z 908.027,A -85,B 0,C 180,E1 -18989.997,E2 -18989.997} C_VEL
LIN {X 0,Y 249.955,Z 907.256,A -85,B 0,C 180,E1 -18993.221,E2 -18993.221} C_VEL
LIN {X 0,Y 250.227,Z 906.312,A -85,B 0,C 180,E1 -18994.83,E2 -18994.83} C_VEL
LIN {X 0,Y 250.362,Z 905.022,A -85,B 0,C 180,E1 -18996.444,E2 -18996.444} C_VEL
LIN {X 0,Y 251.158,Z 902.214,A -85,B 0,C 180,E1 -18998.85,E2 -18998.85} C_VEL
LIN {X 0,Y 252.451,Z 898.368,A -85,B 0,C 180,E1 -19001.234,E2 -19001.234} C_VEL
LIN {X 0,Y 253.766,Z 893.453,A -85,B 0,C 180,E1 -19003.612,E2 -19003.612} C_VEL
LIN {X 0,Y 255.173,Z 887.277,A -85,B 0,C 180,E1 -19005.984,E2 -19005.984} C_VEL
LIN {X 0,Y 257.069,Z 879.499,A -85,B 0,C 180,E1 -19008.321,E2 -19008.321} C_VEL
LIN {X 0,Y 258.833,Z 871.561,A -85,B 0,C 180,E1 -19010.252,E2 -19010.252} C_VEL
LIN {X 0,Y 260.751,Z 861.86,A -85,B 0,C 180,E1 -19012.166,E2 -19012.166} C_VEL
LIN {X 0,Y 261.6,Z 857.142,A -85,B 0,C 180,E1 -19012.954,E2 -19012.954} C_VEL
LIN {X 0,Y 259.22,Z 847.782,A -85,B 0,C 180,E1 -19014.776,E2 -19014.776} C_VEL
LIN {X 0,Y 255.632,Z 837.096,A -85,B 0,C 180,E1 -19016.64,E2 -19016.64} C_VEL
LIN {X 0,Y 251.495,Z 827.038,A -85,B 0,C 180,E1 -19018.236,E2 -19018.236} C_VEL
LIN {X 0,Y 249.225,Z 822.183,A -85,B 0,C 180,E1 -19018.962,E2 -19018.962} C_VEL
LIN {X 0,Y 249.081,Z 821.46,A -85,B 0,C 180,E1 -19019.064,E2 -19019.064} C_VEL
LIN {X 0,Y 249.03,Z 821.467,A -85,B 0,C 180,E1 -19022.422,E2 -19022.422} C_VEL
LIN {X 0,Y 249.069,Z 821.462,A -85,B 0,C 180,E1 -19026.335,E2 -19026.335} C_VEL
LIN {X 0,Y 249.076,Z 821.461,A -85,B 0,C 180,E1 -19030.46,E2 -19030.46} C_VEL
LIN {X 0,Y 249.087,Z 821.458,A -85,B 0,C 180,E1 -19032.811,E2 -19032.811} C_VEL
LIN {X 0,Y 249.089,Z 821.45,A -85,B 0,C 180,E1 -19037.378,E2 -19037.378} C_VEL
LIN {X 0,Y 249.063,Z 821.453,A -85,B 0,C 180,E1 -19041.626,E2 -19041.626} C_VEL
LIN {X 0,Y 249.05,Z 821.453,A -85,B 0,C 180,E1 -19045.64,E2 -19045.64} C_VEL
LIN {X 0,Y 249.039,Z 821.456,A -85,B 0,C 180,E1 -19049.471,E2 -19049.471} C_VEL
LIN {X 0,Y 249.061,Z 821.458,A -85,B 0,C 180,E1 -19053.161,E2 -19053.161} C_VEL
LIN {X 0,Y 249.066,Z 821.461,A -85,B 0,C 180,E1 -19056.731,E2 -19056.731} C_VEL
LIN {X 0,Y 249.096,Z 821.451,A -85,B 0,C 180,E1 -19060.21,E2 -19060.21} C_VEL
LIN {X 0,Y 249.228,Z 821.432,A -85,B 0,C 180,E1 -19063.621,E2 -19063.621} C_VEL
LIN {X 0,Y 249.238,Z 821.441,A -85,B 0,C 180,E1 -19068.616,E2 -19068.616} C_VEL
LIN {X 0,Y 249.464,Z 821.407,A -85,B 0,C 180,E1 -19071.902,E2 -19071.902} C_VEL
LIN {X 0,Y 249.419,Z 821.41,A -85,B 0,C 180,E1 -19076.769,E2 -19076.769} C_VEL
LIN {X 0,Y 249.712,Z 821.384,A -85,B 0,C 180,E1 -19080,E2 -19080} C_VEL
LIN {X 0,Y 249.417,Z 821.421,A -85,B 0,C 180,E1 -19083.231,E2 -19083.231} C_VEL
LIN {X 0,Y 249.46,Z 821.411,A -85,B 0,C 180,E1 -19088.098,E2 -19088.098} C_VEL
LIN {X 0,Y 249.238,Z 821.435,A -85,B 0,C 180,E1 -19091.384,E2 -19091.384} C_VEL
LIN {X 0,Y 249.227,Z 821.443,A -85,B 0,C 180,E1 -19096.379,E2 -19096.379} C_VEL
LIN {X 0,Y 249.069,Z 821.462,A -85,B 0,C 180,E1 -19101.52,E2 -19101.52} C_VEL
LIN {X 0,Y 249.07,Z 821.459,A -85,B 0,C 180,E1 -19105.461,E2 -19105.461} C_VEL
LIN {X 0,Y 249.023,Z 821.467,A -85,B 0,C 180,E1 -19108.975,E2 -19108.975} C_VEL
LIN {X 0,Y 249.024,Z 821.465,A -85,B 0,C 180,E1 -19113.475,E2 -19113.475} C_VEL
LIN {X 0,Y 248.749,Z 822.369,A -85,B 0,C 180,E1 -19114.378,E2 -19114.378} C_VEL
LIN {X 0,Y 247.245,Z 825.365,A -85,B 0,C 180,E1 -19116.066,E2 -19116.066} C_VEL
LIN {X 0,Y 244.328,Z 830.733,A -85,B 0,C 180,E1 -19118.96,E2 -19118.96} C_VEL
LIN {X 0,Y 244.148,Z 832.764,A -85,B 0,C 180,E1 -19120.258,E2 -19120.258} C_VEL
LIN {X 0,Y 245.633,Z 840.1,A -85,B 0,C 180,E1 -19124.847,E2 -19124.847} C_VEL
LIN {X 0,Y 246.957,Z 847.417,A -85,B 0,C 180,E1 -19129.12,E2 -19129.12} C_VEL
LIN {X 0,Y 247.292,Z 850.316,A -85,B 0,C 180,E1 -19130.722,E2 -19130.722} C_VEL
LIN {X 0,Y 245.908,Z 856.957,A -85,B 0,C 180,E1 -19134.139,E2 -19134.139} C_VEL
LIN {X 0,Y 243.803,Z 867.157,A -85,B 0,C 180,E1 -19139.331,E2 -19139.331} C_VEL
LIN {X 0,Y 246.402,Z 881.586,A -85,B 0,C 180,E1 -19140.42,E2 -19140.42} C_VEL
LIN {X 0,Y 247.874,Z 894.776,A -85,B 0,C 180,E1 -19141.654,E2 -19141.654} C_VEL
LIN {X 0,Y 248.563,Z 907.42,A -85,B 0,C 180,E1 -19143.106,E2 -19143.106} C_VEL
LIN {X 0,Y 248.448,Z 920.017,A -85,B 0,C 180,E1 -19144.851,E2 -19144.851} C_VEL
LIN {X 0,Y 247.716,Z 930.456,A -85,B 0,C 180,E1 -19146.601,E2 -19146.601} C_VEL
LIN {X 0,Y 246.782,Z 940.774,A -85,B 0,C 180,E1 -19148.713,E2 -19148.713} C_VEL
LIN {X 0,Y 244.625,Z 950.633,A -85,B 0,C 180,E1 -19151.146,E2 -19151.146} C_VEL
LIN {X 0,Y 243,Z 957.305,A -85,B 0,C 180,E1 -19153.192,E2 -19153.192} C_VEL
LIN {X 0,Y 241.932,Z 963.978,A -85,B 0,C 180,E1 -19155.708,E2 -19155.708} C_VEL
LIN {X 0,Y 241.181,Z 969.304,A -85,B 0,C 180,E1 -19158.233,E2 -19158.233} C_VEL
LIN {X 0,Y 240.925,Z 973.5,A -85,B 0,C 180,E1 -19160.771,E2 -19160.771} C_VEL
LIN {X 0,Y 241.017,Z 976.644,A -85,B 0,C 180,E1 -19163.305,E2 -19163.305} C_VEL
LIN {X 0,Y 241.256,Z 978.168,A -85,B 0,C 180,E1 -19164.989,E2 -19164.989} C_VEL
LIN {X 0,Y 241.476,Z 979.262,A -85,B 0,C 180,E1 -19166.666,E2 -19166.666} C_VEL
LIN {X 0,Y 241.683,Z 979.937,A -85,B 0,C 180,E1 -19168.337,E2 -19168.337} C_VEL
LIN {X 0,Y 241.876,Z 980.191,A -85,B 0,C 180,E1 -19170.003,E2 -19170.003} C_VEL
LIN {X 0,Y 241.685,Z 979.927,A -85,B 0,C 180,E1 -19171.669,E2 -19171.669} C_VEL
LIN {X 0,Y 241.486,Z 979.244,A -85,B 0,C 180,E1 -19173.34,E2 -19173.34} C_VEL
LIN {X 0,Y 241.28,Z 978.145,A -85,B 0,C 180,E1 -19175.016,E2 -19175.016} C_VEL
LIN {X 0,Y 241.021,Z 975.689,A -85,B 0,C 180,E1 -19177.512,E2 -19177.512} C_VEL
LIN {X 0,Y 240.978,Z 972.511,A -85,B 0,C 180,E1 -19180.081,E2 -19180.081} C_VEL
LIN {X 0,Y 241.318,Z 969.804,A -85,B 0,C 180,E1 -19182.619,E2 -19182.619} C_VEL
LIN {X 0,Y 242.261,Z 966.275,A -85,B 0,C 180,E1 -19185.138,E2 -19185.138} C_VEL
LIN {X 0,Y 244.4,Z 960.163,A -85,B 0,C 180,E1 -19188.443,E2 -19188.443} C_VEL
LIN {X 0,Y 247.201,Z 953.402,A -85,B 0,C 180,E1 -19191.256,E2 -19191.256} C_VEL
LIN {X 0,Y 250.17,Z 946.584,A -85,B 0,C 180,E1 -19193.601,E2 -19193.601} C_VEL
LIN {X 0,Y 252.819,Z 938.777,A -85,B 0,C 180,E1 -19195.968,E2 -19195.968} C_VEL
LIN {X 0,Y 256.389,Z 929.081,A -85,B 0,C 180,E1 -19198.467,E2 -19198.467} C_VEL
LIN {X 0,Y 258.701,Z 921.613,A -85,B 0,C 180,E1 -19200.174,E2 -19200.174} C_VEL
LIN {X 0,Y 261.225,Z 909.811,A -85,B 0,C 180,E1 -19202.888,E2 -19202.888} C_VEL
LIN {X 0,Y 263.034,Z 898.8,A -85,B 0,C 180,E1 -19205.437,E2 -19205.437} C_VEL
LIN {X 0,Y 264.287,Z 889.59,A -85,B 0,C 180,E1 -19207.71,E2 -19207.71} C_VEL
LIN {X 0,Y 265.146,Z 882.662,A -85,B 0,C 180,E1 -19209.508,E2 -19209.508} C_VEL
LIN {X 0,Y 265.907,Z 878.184,A -85,B 0,C 180,E1 -19210.726,E2 -19210.726} C_VEL
LIN {X 0,Y 266.519,Z 872.316,A -85,B 0,C 180,E1 -19212.753,E2 -19212.753} C_VEL
LIN {X 0,Y 266.842,Z 868.431,A -85,B 0,C 180,E1 -19214.674,E2 -19214.674} C_VEL
LIN {X 0,Y 267.363,Z 865.063,A -85,B 0,C 180,E1 -19217.396,E2 -19217.396} C_VEL
LIN {X 0,Y 268.094,Z 863.673,A -85,B 0,C 180,E1 -19219.487,E2 -19219.487} C_VEL
LIN {X 0,Y 269.052,Z 863.43,A -85,B 0,C 180,E1 -19221.598,E2 -19221.598} C_VEL
LIN {X 0,Y 270.018,Z 864.406,A -85,B 0,C 180,E1 -19223.794,E2 -19223.794} C_VEL
LIN {X 0,Y 271.269,Z 866.474,A -85,B 0,C 180,E1 -19226.005,E2 -19226.005} C_VEL
LIN {X 0,Y 271.782,Z 869.82,A -85,B 0,C 180,E1 -19228.029,E2 -19228.029} C_VEL
LIN {X 0,Y 272.135,Z 875.173,A -85,B 0,C 180,E1 -19230.615,E2 -19230.615} C_VEL
LIN {X 0,Y 271.928,Z 879.681,A -85,B 0,C 180,E1 -19232.499,E2 -19232.499} C_VEL
LIN {X 0,Y 268.059,Z 887.157,A -85,B 0,C 180,E1 -19234.367,E2 -19234.367} C_VEL
LIN {X 0,Y 263.989,Z 893.864,A -85,B 0,C 180,E1 -19236.463,E2 -19236.463} C_VEL
LIN {X 0,Y 260.276,Z 899.438,A -85,B 0,C 180,E1 -19238.621,E2 -19238.621} C_VEL
LIN {X 0,Y 256.943,Z 903.907,A -85,B 0,C 180,E1 -19240.839,E2 -19240.839} C_VEL
LIN {X 0,Y 253.932,Z 907.43,A -85,B 0,C 180,E1 -19243.106,E2 -19243.106} C_VEL
LIN {X 0,Y 251.247,Z 909.911,A -85,B 0,C 180,E1 -19245.419,E2 -19245.419} C_VEL
LIN {X 0,Y 248.223,Z 911.99,A -85,B 0,C 180,E1 -19248.569,E2 -19248.569} C_VEL
LIN {X 0,Y 245.902,Z 912.415,A -85,B 0,C 180,E1 -19251.784,E2 -19251.784} C_VEL
LIN {X 0,Y 244.959,Z 912.077,A -85,B 0,C 180,E1 -19253.41,E2 -19253.41} C_VEL
LIN {X 0,Y 244.26,Z 911.332,A -85,B 0,C 180,E1 -19255.048,E2 -19255.048} C_VEL
LIN {X 0,Y 243.121,Z 908.617,A -85,B 0,C 180,E1 -19258.344,E2 -19258.344} C_VEL
LIN {X 0,Y 242.454,Z 905.559,A -85,B 0,C 180,E1 -19260.831,E2 -19260.831} C_VEL
LIN {X 0,Y 242.133,Z 901.52,A -85,B 0,C 180,E1 -19263.328,E2 -19263.328} C_VEL
LIN {X 0,Y 242.355,Z 895.475,A -85,B 0,C 180,E1 -19266.243,E2 -19266.243} C_VEL
LIN {X 0,Y 242.841,Z 888.918,A -85,B 0,C 180,E1 -19268.739,E2 -19268.739} C_VEL
LIN {X 0,Y 243.419,Z 880.646,A -85,B 0,C 180,E1 -19271.345,E2 -19271.345} C_VEL
LIN {X 0,Y 244.145,Z 873.002,A -85,B 0,C 180,E1 -19273.314,E2 -19273.314} C_VEL
LIN {X 0,Y 244.952,Z 864.621,A -85,B 0,C 180,E1 -19275.178,E2 -19275.178} C_VEL
LIN {X 0,Y 245.719,Z 855.908,A -85,B 0,C 180,E1 -19276.834,E2 -19276.834} C_VEL
LIN {X 0,Y 246.759,Z 845.387,A -85,B 0,C 180,E1 -19278.536,E2 -19278.536} C_VEL
LIN {X 0,Y 246.813,Z 842.184,A -85,B 0,C 180,E1 -19278.998,E2 -19278.998} C_VEL
LIN {X 0,Y 243.714,Z 829.502,A -85,B 0,C 180,E1 -19280.715,E2 -19280.715} C_VEL
LIN {X 0,Y 242.031,Z 822.323,A -85,B 0,C 180,E1 -19281.587,E2 -19281.587} C_VEL
LIN {X 0,Y 241.995,Z 822.333,A -85,B 0,C 180,E1 -19285.826,E2 -19285.826} C_VEL
LIN {X 0,Y 241.971,Z 822.34,A -85,B 0,C 180,E1 -19289.588,E2 -19289.588} C_VEL
LIN {X 0,Y 241.987,Z 822.329,A -85,B 0,C 180,E1 -19293.492,E2 -19293.492} C_VEL
LIN {X 0,Y 241.991,Z 822.33,A -85,B 0,C 180,E1 -19297.582,E2 -19297.582} C_VEL
LIN {X 0,Y 241.916,Z 822.343,A -85,B 0,C 180,E1 -19301.927,E2 -19301.927} C_VEL
LIN {X 0,Y 241.907,Z 822.346,A -85,B 0,C 180,E1 -19306.579,E2 -19306.579} C_VEL
LIN {X 0,Y 241.991,Z 822.342,A -85,B 0,C 180,E1 -19311.642,E2 -19311.642} C_VEL
LIN {X 0,Y 241.981,Z 822.344,A -85,B 0,C 180,E1 -19314.485,E2 -19314.485} C_VEL
LIN {X 0,Y 241.98,Z 822.335,A -85,B 0,C 180,E1 -19318.478,E2 -19318.478} C_VEL
LIN {X 0,Y 242.017,Z 822.332,A -85,B 0,C 180,E1 -19320.116,E2 -19320.116} C_VEL
LIN {X 0,Y 243.144,Z 825.318,A -85,B 0,C 180,E1 -19320.55,E2 -19320.55} C_VEL
LIN {X 0,Y 247.519,Z 834.89,A -85,B 0,C 180,E1 -19322.13,E2 -19322.13} C_VEL
LIN {X 0,Y 251.282,Z 845.254,A -85,B 0,C 180,E1 -19323.961,E2 -19323.961} C_VEL
LIN {X 0,Y 254.087,Z 855.155,A -85,B 0,C 180,E1 -19325.892,E2 -19325.892} C_VEL
LIN {X 0,Y 254.879,Z 858.564,A -85,B 0,C 180,E1 -19326.604,E2 -19326.604} C_VEL
LIN {X 0,Y 253.035,Z 868.354,A -85,B 0,C 180,E1 -19328.404,E2 -19328.404} C_VEL
LIN {X 0,Y 251.237,Z 877.032,A -85,B 0,C 180,E1 -19330.383,E2 -19330.383} C_VEL
LIN {X 0,Y 249.367,Z 884.219,A -85,B 0,C 180,E1 -19332.361,E2 -19332.361} C_VEL
LIN {X 0,Y 247.783,Z 890.901,A -85,B 0,C 180,E1 -19334.658,E2 -19334.658} C_VEL
LIN {X 0,Y 246.552,Z 895.951,A -85,B 0,C 180,E1 -19336.815,E2 -19336.815} C_VEL
LIN {X 0,Y 245.007,Z 900.588,A -85,B 0,C 180,E1 -19339.251,E2 -19339.251} C_VEL
LIN {X 0,Y 243.925,Z 904.11,A -85,B 0,C 180,E1 -19341.714,E2 -19341.714} C_VEL
LIN {X 0,Y 243.448,Z 905.917,A -85,B 0,C 180,E1 -19343.366,E2 -19343.366} C_VEL
LIN {X 0,Y 243.242,Z 907.252,A -85,B 0,C 180,E1 -19345.025,E2 -19345.025} C_VEL
LIN {X 0,Y 242.714,Z 908.83,A -85,B 0,C 180,E1 -19348.338,E2 -19348.338} C_VEL
LIN {X 0,Y 242.64,Z 909.058,A -85,B 0,C 180,E1 -19349.997,E2 -19349.997} C_VEL
LIN {X 0,Y 242.942,Z 908.287,A -85,B 0,C 180,E1 -19353.314,E2 -19353.314} C_VEL
LIN {X 0,Y 243.228,Z 907.342,A -85,B 0,C 180,E1 -19354.97,E2 -19354.97} C_VEL
LIN {X 0,Y 243.382,Z 906.053,A -85,B 0,C 180,E1 -19356.63,E2 -19356.63} C_VEL
LIN {X 0,Y 244.219,Z 903.245,A -85,B 0,C 180,E1 -19359.104,E2 -19359.104} C_VEL
LIN {X 0,Y 245.565,Z 899.398,A -85,B 0,C 180,E1 -19361.554,E2 -19361.554} C_VEL
LIN {X 0,Y 246.946,Z 894.482,A -85,B 0,C 180,E1 -19363.996,E2 -19363.996} C_VEL
LIN {X 0,Y 248.426,Z 888.306,A -85,B 0,C 180,E1 -19366.43,E2 -19366.43} C_VEL
LIN {X 0,Y 250.413,Z 880.527,A -85,B 0,C 180,E1 -19368.826,E2 -19368.826} C_VEL
LIN {X 0,Y 252.257,Z 872.589,A -85,B 0,C 180,E1 -19370.804,E2 -19370.804} C_VEL
LIN {X 0,Y 254.271,Z 862.886,A -85,B 0,C 180,E1 -19372.762,E2 -19372.762} C_VEL
LIN {X 0,Y 255.002,Z 858.786,A -85,B 0,C 180,E1 -19373.469,E2 -19373.469} C_VEL
LIN {X 0,Y 252.644,Z 849.562,A -85,B 0,C 180,E1 -19375.354,E2 -19375.354} C_VEL
LIN {X 0,Y 249.23,Z 839.369,A -85,B 0,C 180,E1 -19377.236,E2 -19377.236} C_VEL
LIN {X 0,Y 244.999,Z 829.079,A -85,B 0,C 180,E1 -19378.966,E2 -19378.966} C_VEL
LIN {X 0,Y 242.209,Z 823.265,A -85,B 0,C 180,E1 -19379.892,E2 -19379.892} C_VEL
LIN {X 0,Y 242.022,Z 822.34,A -85,B 0,C 180,E1 -19380.056,E2 -19380.056} C_VEL
LIN {X 0,Y 241.985,Z 822.343,A -85,B 0,C 180,E1 -19383.488,E2 -19383.488} C_VEL
LIN {X 0,Y 242.006,Z 822.341,A -85,B 0,C 180,E1 -19387.574,E2 -19387.574} C_VEL
LIN {X 0,Y 242.03,Z 822.338,A -85,B 0,C 180,E1 -19391.898,E2 -19391.898} C_VEL
LIN {X 0,Y 242.015,Z 822.334,A -85,B 0,C 180,E1 -19396.546,E2 -19396.546} C_VEL
LIN {X 0,Y 242.018,Z 822.336,A -85,B 0,C 180,E1 -19400.293,E2 -19400.293} C_VEL
LIN {X 0,Y 242.025,Z 822.334,A -85,B 0,C 180,E1 -19404.495,E2 -19404.495} C_VEL
LIN {X 0,Y 241.964,Z 822.344,A -85,B 0,C 180,E1 -19408.478,E2 -19408.478} C_VEL
LIN {X 0,Y 241.996,Z 822.341,A -85,B 0,C 180,E1 -19412.311,E2 -19412.311} C_VEL
LIN {X 0,Y 242.044,Z 822.332,A -85,B 0,C 180,E1 -19416.014,E2 -19416.014} C_VEL
LIN {X 0,Y 242.023,Z 822.331,A -85,B 0,C 180,E1 -19419.607,E2 -19419.607} C_VEL
LIN {X 0,Y 242.149,Z 822.315,A -85,B 0,C 180,E1 -19423.277,E2 -19423.277} C_VEL
LIN {X 0,Y 242.172,Z 822.32,A -85,B 0,C 180,E1 -19428.279,E2 -19428.279} C_VEL
LIN {X 0,Y 242.411,Z 822.283,A -85,B 0,C 180,E1 -19431.665,E2 -19431.665} C_VEL
LIN {X 0,Y 242.243,Z 822.314,A -85,B 0,C 180,E1 -19435.007,E2 -19435.007} C_VEL
LIN {X 0,Y 242.621,Z 822.265,A -85,B 0,C 180,E1 -19438.34,E2 -19438.34} C_VEL
LIN {X 0,Y 242.62,Z 822.268,A -85,B 0,C 180,E1 -19441.66,E2 -19441.66} C_VEL
LIN {X 0,Y 242.41,Z 822.288,A -85,B 0,C 180,E1 -19446.659,E2 -19446.659} C_VEL
LIN {X 0,Y 242.299,Z 822.304,A -85,B 0,C 180,E1 -19450.022,E2 -19450.022} C_VEL
LIN {X 0,Y 242.152,Z 822.323,A -85,B 0,C 180,E1 -19455.142,E2 -19455.142} C_VEL
LIN {X 0,Y 242.057,Z 822.336,A -85,B 0,C 180,E1 -19458.625,E2 -19458.625} C_VEL
LIN {X 0,Y 241.99,Z 822.344,A -85,B 0,C 180,E1 -19462.182,E2 -19462.182} C_VEL
LIN {X 0,Y 242.018,Z 822.339,A -85,B 0,C 180,E1 -19465.823,E2 -19465.823} C_VEL
LIN {X 0,Y 241.955,Z 822.345,A -85,B 0,C 180,E1 -19469.59,E2 -19469.59} C_VEL
LIN {X 0,Y 241.987,Z 822.409,A -85,B 0,C 180,E1 -19472.98,E2 -19472.98} C_VEL
LIN {X 0,Y 243.288,Z 828.432,A -85,B 0,C 180,E1 -19477.347,E2 -19477.347} C_VEL
LIN {X 0,Y 244.148,Z 832.764,A -85,B 0,C 180,E1 -19480.258,E2 -19480.258} C_VEL
LIN {X 0,Y 243.917,Z 834.934,A -85,B 0,C 180,E1 -19481.546,E2 -19481.546} C_VEL
LIN {X 0,Y 241.775,Z 838.914,A -85,B 0,C 180,E1 -19483.629,E2 -19483.629} C_VEL
LIN {X 0,Y 239.917,Z 842.182,A -85,B 0,C 180,E1 -19485.314,E2 -19485.314} C_VEL
LIN {X 0,Y 239.308,Z 844.539,A -85,B 0,C 180,E1 -19486.619,E2 -19486.619} C_VEL
LIN {X 0,Y 239.368,Z 845.286,A -85,B 0,C 180,E1 -19487.061,E2 -19487.061} C_VEL
LIN {X 0,Y 240.221,Z 850.168,A -85,B 0,C 180,E1 -19489.941,E2 -19489.941} C_VEL
LIN {X 0,Y 240.189,Z 852.122,A -85,B 0,C 180,E1 -19491.021,E2 -19491.021} C_VEL
LIN {X 0,Y 238.455,Z 859.536,A -85,B 0,C 180,E1 -19494.925,E2 -19494.925} C_VEL
LIN {X 0,Y 237.054,Z 866.001,A -85,B 0,C 180,E1 -19498.35,E2 -19498.35} C_VEL
LIN {X 0,Y 239.778,Z 881.158,A -85,B 0,C 180,E1 -19499.563,E2 -19499.563} C_VEL
LIN {X 0,Y 241.263,Z 894.766,A -85,B 0,C 180,E1 -19500.915,E2 -19500.915} C_VEL
LIN {X 0,Y 241.884,Z 906.323,A -85,B 0,C 180,E1 -19502.301,E2 -19502.301} C_VEL
LIN {X 0,Y 241.788,Z 917.752,A -85,B 0,C 180,E1 -19503.923,E2 -19503.923} C_VEL
LIN {X 0,Y 241.116,Z 928.39,A -85,B 0,C 180,E1 -19505.724,E2 -19505.724} C_VEL
LIN {X 0,Y 240.102,Z 937.825,A -85,B 0,C 180,E1 -19507.638,E2 -19507.638} C_VEL
LIN {X 0,Y 239.353,Z 943.261,A -85,B 0,C 180,E1 -19508.922,E2 -19508.922} C_VEL
LIN {X 0,Y 237.51,Z 950.993,A -85,B 0,C 180,E1 -19511.008,E2 -19511.008} C_VEL
LIN {X 0,Y 235.906,Z 957.454,A -85,B 0,C 180,E1 -19513.118,E2 -19513.118} C_VEL
LIN {X 0,Y 234.974,Z 962.924,A -85,B 0,C 180,E1 -19515.275,E2 -19515.275} C_VEL
LIN {X 0,Y 234.179,Z 968.255,A -85,B 0,C 180,E1 -19517.876,E2 -19517.876} C_VEL
LIN {X 0,Y 233.87,Z 972.451,A -85,B 0,C 180,E1 -19520.49,E2 -19520.49} C_VEL
LIN {X 0,Y 233.955,Z 975.6,A -85,B 0,C 180,E1 -19523.102,E2 -19523.102} C_VEL
LIN {X 0,Y 234.19,Z 977.127,A -85,B 0,C 180,E1 -19524.838,E2 -19524.838} C_VEL
LIN {X 0,Y 234.418,Z 978.224,A -85,B 0,C 180,E1 -19526.566,E2 -19526.566} C_VEL
LIN {X 0,Y 234.636,Z 978.903,A -85,B 0,C 180,E1 -19528.287,E2 -19528.287} C_VEL
LIN {X 0,Y 234.844,Z 979.158,A -85,B 0,C 180,E1 -19530.003,E2 -19530.003} C_VEL
LIN {X 0,Y 234.639,Z 978.892,A -85,B 0,C 180,E1 -19531.719,E2 -19531.719} C_VEL
LIN {X 0,Y 234.429,Z 978.206,A -85,B 0,C 180,E1 -19533.44,E2 -19533.44} C_VEL
LIN {X 0,Y 234.214,Z 977.103,A -85,B 0,C 180,E1 -19535.168,E2 -19535.168} C_VEL
LIN {X 0,Y 233.97,Z 974.819,A -85,B 0,C 180,E1 -19537.581,E2 -19537.581} C_VEL
LIN {X 0,Y 234.96,Z 966.834,A -85,B 0,C 180,E1 -19544.732,E2 -19544.732} C_VEL
LIN {X 0,Y 236.431,Z 962.932,A -85,B 0,C 180,E1 -19547.296,E2 -19547.296} C_VEL
LIN {X 0,Y 238.444,Z 958.248,A -85,B 0,C 180,E1 -19549.816,E2 -19549.816} C_VEL
LIN {X 0,Y 241.099,Z 952.525,A -85,B 0,C 180,E1 -19552.271,E2 -19552.271} C_VEL
LIN {X 0,Y 243.661,Z 947.135,A -85,B 0,C 180,E1 -19554.272,E2 -19554.272} C_VEL
LIN {X 0,Y 247.047,Z 938.364,A -85,B 0,C 180,E1 -19557.079,E2 -19557.079} C_VEL
LIN {X 0,Y 251.796,Z 926.716,A -85,B 0,C 180,E1 -19560.162,E2 -19560.162} C_VEL
LIN {X 0,Y 254.582,Z 916.965,A -85,B 0,C 180,E1 -19562.572,E2 -19562.572} C_VEL
LIN {X 0,Y 256.996,Z 906.853,A -85,B 0,C 180,E1 -19565.052,E2 -19565.052} C_VEL
LIN {X 0,Y 259.141,Z 896.105,A -85,B 0,C 180,E1 -19567.79,E2 -19567.79} C_VEL
LIN {X 0,Y 260.904,Z 887.113,A -85,B 0,C 180,E1 -19570.28,E2 -19570.28} C_VEL
LIN {X 0,Y 262.099,Z 881.015,A -85,B 0,C 180,E1 -19572.098,E2 -19572.098} C_VEL
LIN {X 0,Y 262.622,Z 878.322,A -85,B 0,C 180,E1 -19573.055,E2 -19573.055} C_VEL
LIN {X 0,Y 263.114,Z 875.245,A -85,B 0,C 180,E1 -19574.488,E2 -19574.488} C_VEL
LIN {X 0,Y 263.44,Z 872.893,A -85,B 0,C 180,E1 -19576.082,E2 -19576.082} C_VEL
LIN {X 0,Y 264.061,Z 870.622,A -85,B 0,C 180,E1 -19578.289,E2 -19578.289} C_VEL
LIN {X 0,Y 264.805,Z 869.603,A -85,B 0,C 180,E1 -19580.434,E2 -19580.434} C_VEL
LIN {X 0,Y 265.666,Z 869.765,A -85,B 0,C 180,E1 -19582.529,E2 -19582.529} C_VEL
LIN {X 0,Y 266.593,Z 871.126,A -85,B 0,C 180,E1 -19584.812,E2 -19584.812} C_VEL
LIN {X 0,Y 267.084,Z 872.995,A -85,B 0,C 180,E1 -19586.455,E2 -19586.455} C_VEL
LIN {X 0,Y 267.204,Z 877.73,A -85,B 0,C 180,E1 -19589.176,E2 -19589.176} C_VEL
LIN {X 0,Y 266.786,Z 882.995,A -85,B 0,C 180,E1 -19591.694,E2 -19591.694} C_VEL
LIN {X 0,Y 262.315,Z 890.726,A -85,B 0,C 180,E1 -19593.764,E2 -19593.764} C_VEL
LIN {X 0,Y 256.72,Z 898.91,A -85,B 0,C 180,E1 -19596.612,E2 -19596.612} C_VEL
LIN {X 0,Y 252.933,Z 903.738,A -85,B 0,C 180,E1 -19598.825,E2 -19598.825} C_VEL
LIN {X 0,Y 249.592,Z 907.587,A -85,B 0,C 180,E1 -19601.106,E2 -19601.106} C_VEL
LIN {X 0,Y 246.485,Z 910.43,A -85,B 0,C 180,E1 -19603.433,E2 -19603.433} C_VEL
LIN {X 0,Y 244.664,Z 911.91,A -85,B 0,C 180,E1 -19605.017,E2 -19605.017} C_VEL
LIN {X 0,Y 241.449,Z 913.56,A -85,B 0,C 180,E1 -19608.244,E2 -19608.244} C_VEL
LIN {X 0,Y 240.029,Z 913.862,A -85,B 0,C 180,E1 -19609.882,E2 -19609.882} C_VEL
LIN {X 0,Y 239.011,Z 913.762,A -85,B 0,C 180,E1 -19611.546,E2 -19611.546} C_VEL
LIN {X 0,Y 238.006,Z 913.259,A -85,B 0,C 180,E1 -19613.217,E2 -19613.217} C_VEL
LIN {X 0,Y 237.281,Z 912.347,A -85,B 0,C 180,E1 -19614.902,E2 -19614.902} C_VEL
LIN {X 0,Y 236.078,Z 909.423,A -85,B 0,C 180,E1 -19618.294,E2 -19618.294} C_VEL
LIN {X 0,Y 235.392,Z 906.156,A -85,B 0,C 180,E1 -19620.855,E2 -19620.855} C_VEL
LIN {X 0,Y 235.058,Z 901.894,A -85,B 0,C 180,E1 -19623.428,E2 -19623.428} C_VEL
LIN {X 0,Y 235.297,Z 895.465,A -85,B 0,C 180,E1 -19626.431,E2 -19626.431} C_VEL
LIN {X 0,Y 235.714,Z 889.935,A -85,B 0,C 180,E1 -19628.574,E2 -19628.574} C_VEL
LIN {X 0,Y 236.208,Z 882.778,A -85,B 0,C 180,E1 -19630.917,E2 -19630.917} C_VEL
LIN {X 0,Y 236.855,Z 875.714,A -85,B 0,C 180,E1 -19632.858,E2 -19632.858} C_VEL
LIN {X 0,Y 237.695,Z 866.582,A -85,B 0,C 180,E1 -19634.994,E2 -19634.994} C_VEL
LIN {X 0,Y 238.498,Z 858.035,A -85,B 0,C 180,E1 -19636.697,E2 -19636.697} C_VEL
LIN {X 0,Y 239.635,Z 846.747,A -85,B 0,C 180,E1 -19638.599,E2 -19638.599} C_VEL
LIN {X 0,Y 239.875,Z 844.054,A -85,B 0,C 180,E1 -19638.993,E2 -19638.993} C_VEL
LIN {X 0,Y 236.73,Z 830.654,A -85,B 0,C 180,E1 -19640.87,E2 -19640.87} C_VEL
LIN {X 0,Y 234.985,Z 823.201,A -85,B 0,C 180,E1 -19641.791,E2 -19641.791} C_VEL
LIN {X 0,Y 234.913,Z 823.211,A -85,B 0,C 180,E1 -19646.664,E2 -19646.664} C_VEL
LIN {X 0,Y 234.903,Z 823.22,A -85,B 0,C 180,E1 -19650.572,E2 -19650.572} C_VEL
LIN {X 0,Y 234.931,Z 823.217,A -85,B 0,C 180,E1 -19654.638,E2 -19654.638} C_VEL
LIN {X 0,Y 234.92,Z 823.217,A -85,B 0,C 180,E1 -19658.934,E2 -19658.934} C_VEL
LIN {X 0,Y 234.861,Z 823.226,A -85,B 0,C 180,E1 -19663.492,E2 -19663.492} C_VEL
LIN {X 0,Y 234.859,Z 823.224,A -85,B 0,C 180,E1 -19666.504,E2 -19666.504} C_VEL
LIN {X 0,Y 234.925,Z 823.222,A -85,B 0,C 180,E1 -19671.077,E2 -19671.077} C_VEL
LIN {X 0,Y 234.93,Z 823.22,A -85,B 0,C 180,E1 -19675.359,E2 -19675.359} C_VEL
LIN {X 0,Y 234.976,Z 823.366,A -85,B 0,C 180,E1 -19679.137,E2 -19679.137} C_VEL
LIN {X 0,Y 236.125,Z 826.289,A -85,B 0,C 180,E1 -19679.564,E2 -19679.564} C_VEL
LIN {X 0,Y 241.135,Z 837.167,A -85,B 0,C 180,E1 -19681.47,E2 -19681.47} C_VEL
LIN {X 0,Y 244.336,Z 845.884,A -85,B 0,C 180,E1 -19683.085,E2 -19683.085} C_VEL
LIN {X 0,Y 247.168,Z 855.613,A -85,B 0,C 180,E1 -19685.051,E2 -19685.051} C_VEL
LIN {X 0,Y 248.272,Z 860.231,A -85,B 0,C 180,E1 -19686.062,E2 -19686.062} C_VEL
LIN {X 0,Y 246.98,Z 867.455,A -85,B 0,C 180,E1 -19687.406,E2 -19687.406} C_VEL
LIN {X 0,Y 245.031,Z 876.473,A -85,B 0,C 180,E1 -19689.427,E2 -19689.427} C_VEL
LIN {X 0,Y 242.683,Z 885.253,A -85,B 0,C 180,E1 -19691.859,E2 -19691.859} C_VEL
LIN {X 0,Y 241.016,Z 891.926,A -85,B 0,C 180,E1 -19694.213,E2 -19694.213} C_VEL
LIN {X 0,Y 239.718,Z 896.984,A -85,B 0,C 180,E1 -19696.432,E2 -19696.432} C_VEL
LIN {X 0,Y 238.11,Z 901.621,A -85,B 0,C 180,E1 -19698.936,E2 -19698.936} C_VEL
LIN {X 0,Y 236.976,Z 905.142,A -85,B 0,C 180,E1 -19701.47,E2 -19701.47} C_VEL
LIN {X 0,Y 236.491,Z 906.946,A -85,B 0,C 180,E1 -19703.17,E2 -19703.17} C_VEL
LIN {X 0,Y 236.248,Z 908.283,A -85,B 0,C 180,E1 -19704.877,E2 -19704.877} C_VEL
LIN {X 0,Y 235.693,Z 909.861,A -85,B 0,C 180,E1 -19708.288,E2 -19708.288} C_VEL
LIN {X 0,Y 235.616,Z 910.089,A -85,B 0,C 180,E1 -19709.997,E2 -19709.997} C_VEL
LIN {X 0,Y 235.929,Z 909.318,A -85,B 0,C 180,E1 -19713.412,E2 -19713.412} C_VEL
LIN {X 0,Y 236.231,Z 908.373,A -85,B 0,C 180,E1 -19715.117,E2 -19715.117} C_VEL
LIN {X 0,Y 236.405,Z 907.084,A -85,B 0,C 180,E1 -19716.826,E2 -19716.826} C_VEL
LIN {X 0,Y 237.284,Z 904.275,A -85,B 0,C 180,E1 -19719.372,E2 -19719.372} C_VEL
LIN {X 0,Y 238.686,Z 900.428,A -85,B 0,C 180,E1 -19721.891,E2 -19721.891} C_VEL
LIN {X 0,Y 240.137,Z 895.512,A -85,B 0,C 180,E1 -19724.401,E2 -19724.401} C_VEL
LIN {X 0,Y 241.722,Z 889.331,A -85,B 0,C 180,E1 -19726.899,E2 -19726.899} C_VEL
LIN {X 0,Y 243.777,Z 881.555,A -85,B 0,C 180,E1 -19729.359,E2 -19729.359} C_VEL
LIN {X 0,Y 245.704,Z 873.617,A -85,B 0,C 180,E1 -19731.385,E2 -19731.385} C_VEL
LIN {X 0,Y 247.809,Z 863.914,A -85,B 0,C 180,E1 -19733.39,E2 -19733.39} C_VEL
LIN {X 0,Y 248.369,Z 860.404,A -85,B 0,C 180,E1 -19734.024,E2 -19734.024} C_VEL
LIN {X 0,Y 246.116,Z 851.577,A -85,B 0,C 180,E1 -19735.916,E2 -19735.916} C_VEL
LIN {X 0,Y 243.162,Z 842.531,A -85,B 0,C 180,E1 -19737.685,E2 -19737.685} C_VEL
LIN {X 0,Y 239.708,Z 833.66,A -85,B 0,C 180,E1 -19739.28,E2 -19739.28} C_VEL
LIN {X 0,Y 235.057,Z 823.891,A -85,B 0,C 180,E1 -19740.948,E2 -19740.948} C_VEL
LIN {X 0,Y 234.943,Z 823.221,A -85,B 0,C 180,E1 -19741.061,E2 -19741.061} C_VEL
LIN {X 0,Y 234.954,Z 823.219,A -85,B 0,C 180,E1 -19744.63,E2 -19744.63} C_VEL
LIN {X 0,Y 234.959,Z 823.218,A -85,B 0,C 180,E1 -19748.949,E2 -19748.949} C_VEL
LIN {X 0,Y 234.989,Z 823.214,A -85,B 0,C 180,E1 -19753.457,E2 -19753.457} C_VEL
LIN {X 0,Y 234.993,Z 823.209,A -85,B 0,C 180,E1 -19758.384,E2 -19758.384} C_VEL
LIN {X 0,Y 234.975,Z 823.208,A -85,B 0,C 180,E1 -19761.09,E2 -19761.09} C_VEL
LIN {X 0,Y 234.949,Z 823.21,A -85,B 0,C 180,E1 -19765.365,E2 -19765.365} C_VEL
LIN {X 0,Y 234.957,Z 823.209,A -85,B 0,C 180,E1 -19770.155,E2 -19770.155} C_VEL
LIN {X 0,Y 234.981,Z 823.21,A -85,B 0,C 180,E1 -19773.792,E2 -19773.792} C_VEL
LIN {X 0,Y 234.998,Z 823.206,A -85,B 0,C 180,E1 -19778.968,E2 -19778.968} C_VEL
LIN {X 0,Y 235.082,Z 823.197,A -85,B 0,C 180,E1 -19783.058,E2 -19783.058} C_VEL
LIN {X 0,Y 235.132,Z 823.197,A -85,B 0,C 180,E1 -19787.923,E2 -19787.923} C_VEL
LIN {X 0,Y 235.361,Z 823.16,A -85,B 0,C 180,E1 -19791.413,E2 -19791.413} C_VEL
LIN {X 0,Y 235.387,Z 823.167,A -85,B 0,C 180,E1 -19793.141,E2 -19793.141} C_VEL
LIN {X 0,Y 235.581,Z 823.142,A -85,B 0,C 180,E1 -19798.29,E2 -19798.29} C_VEL
LIN {X 0,Y 235.579,Z 823.145,A -85,B 0,C 180,E1 -19801.709,E2 -19801.709} C_VEL
LIN {X 0,Y 235.382,Z 823.164,A -85,B 0,C 180,E1 -19806.859,E2 -19806.859} C_VEL
LIN {X 0,Y 235.223,Z 823.184,A -85,B 0,C 180,E1 -19810.327,E2 -19810.327} C_VEL
LIN {X 0,Y 235.099,Z 823.201,A -85,B 0,C 180,E1 -19815.607,E2 -19815.607} C_VEL
LIN {X 0,Y 234.992,Z 823.216,A -85,B 0,C 180,E1 -19819.207,E2 -19819.207} C_VEL
LIN {X 0,Y 234.932,Z 823.222,A -85,B 0,C 180,E1 -19822.886,E2 -19822.886} C_VEL
LIN {X 0,Y 234.931,Z 823.218,A -85,B 0,C 180,E1 -19826.662,E2 -19826.662} C_VEL
LIN {X 0,Y 234.923,Z 823.224,A -85,B 0,C 180,E1 -19831.57,E2 -19831.57} C_VEL
LIN {X 0,Y 234.92,Z 823.314,A -85,B 0,C 180,E1 -19832.074,E2 -19832.074} C_VEL
LIN {X 0,Y 236.238,Z 829.238,A -85,B 0,C 180,E1 -19836.566,E2 -19836.566} C_VEL
LIN {X 0,Y 237.687,Z 836.418,A -85,B 0,C 180,E1 -19841.511,E2 -19841.511} C_VEL
LIN {X 0,Y 239.087,Z 843.643,A -85,B 0,C 180,E1 -19846.068,E2 -19846.068} C_VEL
LIN {X 0,Y 239.368,Z 845.286,A -85,B 0,C 180,E1 -19847.061,E2 -19847.061} C_VEL
LIN {X 0,Y 239.036,Z 847.604,A -85,B 0,C 180,E1 -19848.358,E2 -19848.358} C_VEL
LIN {X 0,Y 237.62,Z 850.078,A -85,B 0,C 180,E1 -19849.614,E2 -19849.614} C_VEL
LIN {X 0,Y 232.54,Z 856.878,A -85,B 0,C 180,E1 -19852.972,E2 -19852.972} C_VEL
LIN {X 0,Y 231.832,Z 858.558,A -85,B 0,C 180,E1 -19853.864,E2 -19853.864} C_VEL
LIN {X 0,Y 230.336,Z 864.877,A -85,B 0,C 180,E1 -19857.312,E2 -19857.312} C_VEL
LIN {X 0,Y 233.13,Z 880.199,A -85,B 0,C 180,E1 -19858.61,E2 -19858.61} C_VEL
LIN {X 0,Y 234.572,Z 892.662,A -85,B 0,C 180,E1 -19859.898,E2 -19859.898} C_VEL
LIN {X 0,Y 235.207,Z 905.217,A -85,B 0,C 180,E1 -19861.444,E2 -19861.444} C_VEL
LIN {X 0,Y 235.108,Z 916.661,A -85,B 0,C 180,E1 -19863.124,E2 -19863.124} C_VEL
LIN {X 0,Y 234.494,Z 926.617,A -85,B 0,C 180,E1 -19864.857,E2 -19864.857} C_VEL
LIN {X 0,Y 233.342,Z 936.752,A -85,B 0,C 180,E1 -19866.953,E2 -19866.953} C_VEL
LIN {X 0,Y 232.255,Z 943.873,A -85,B 0,C 180,E1 -19868.712,E2 -19868.712} C_VEL
LIN {X 0,Y 230.053,Z 952.613,A -85,B 0,C 180,E1 -19871.269,E2 -19871.269} C_VEL
LIN {X 0,Y 228.628,Z 958.722,A -85,B 0,C 180,E1 -19873.484,E2 -19873.484} C_VEL
LIN {X 0,Y 227.695,Z 963.766,A -85,B 0,C 180,E1 -19875.708,E2 -19875.708} C_VEL
LIN {X 0,Y 226.991,Z 968.71,A -85,B 0,C 180,E1 -19878.393,E2 -19878.393} C_VEL
LIN {X 0,Y 226.809,Z 972.55,A -85,B 0,C 180,E1 -19881.09,E2 -19881.09} C_VEL
LIN {X 0,Y 226.9,Z 974.557,A -85,B 0,C 180,E1 -19882.886,E2 -19882.886} C_VEL
LIN {X 0,Y 227.126,Z 976.086,A -85,B 0,C 180,E1 -19884.677,E2 -19884.677} C_VEL
LIN {X 0,Y 227.36,Z 977.186,A -85,B 0,C 180,E1 -19886.459,E2 -19886.459} C_VEL
LIN {X 0,Y 227.588,Z 977.867,A -85,B 0,C 180,E1 -19888.234,E2 -19888.234} C_VEL
LIN {X 0,Y 227.812,Z 978.126,A -85,B 0,C 180,E1 -19890.003,E2 -19890.003} C_VEL
LIN {X 0,Y 227.591,Z 977.856,A -85,B 0,C 180,E1 -19891.773,E2 -19891.773} C_VEL
LIN {X 0,Y 227.372,Z 977.168,A -85,B 0,C 180,E1 -19893.547,E2 -19893.547} C_VEL
LIN {X 0,Y 227.151,Z 976.061,A -85,B 0,C 180,E1 -19895.329,E2 -19895.329} C_VEL
LIN {X 0,Y 226.902,Z 973.981,A -85,B 0,C 180,E1 -19897.624,E2 -19897.624} C_VEL
LIN {X 0,Y 226.893,Z 970.612,A -85,B 0,C 180,E1 -19900.714,E2 -19900.714} C_VEL
LIN {X 0,Y 227.669,Z 967.318,A -85,B 0,C 180,E1 -19904.3,E2 -19904.3} C_VEL
LIN {X 0,Y 229.595,Z 962.559,A -85,B 0,C 180,E1 -19907.828,E2 -19907.828} C_VEL
LIN {X 0,Y 232.582,Z 956.401,A -85,B 0,C 180,E1 -19911.263,E2 -19911.263} C_VEL
LIN {X 0,Y 236.16,Z 949.622,A -85,B 0,C 180,E1 -19914.157,E2 -19914.157} C_VEL
LIN {X 0,Y 239.121,Z 942.94,A -85,B 0,C 180,E1 -19916.632,E2 -19916.632} C_VEL
LIN {X 0,Y 242.65,Z 935.318,A -85,B 0,C 180,E1 -19919.025,E2 -19919.025} C_VEL
LIN {X 0,Y 246.403,Z 926.829,A -85,B 0,C 180,E1 -19921.371,E2 -19921.371} C_VEL
LIN {X 0,Y 249.889,Z 916.062,A -85,B 0,C 180,E1 -19924.231,E2 -19924.231} C_VEL
LIN {X 0,Y 252.581,Z 906.576,A -85,B 0,C 180,E1 -19926.745,E2 -19926.745} C_VEL
LIN {X 0,Y 255.567,Z 894.822,A -85,B 0,C 180,E1 -19930.042,E2 -19930.042} C_VEL
LIN {X 0,Y 257.874,Z 886.349,A -85,B 0,C 180,E1 -19932.621,E2 -19932.621} C_VEL
LIN {X 0,Y 258.968,Z 882.17,A -85,B 0,C 180,E1 -19934.287,E2 -19934.287} C_VEL
LIN {X 0,Y 259.355,Z 880.392,A -85,B 0,C 180,E1 -19935.207,E2 -19935.207} C_VEL
LIN {X 0,Y 260.016,Z 877.472,A -85,B 0,C 180,E1 -19937.489,E2 -19937.489} C_VEL
LIN {X 0,Y 260.686,Z 875.981,A -85,B 0,C 180,E1 -19939.682,E2 -19939.682} C_VEL
LIN {X 0,Y 261.355,Z 875.585,A -85,B 0,C 180,E1 -19941.794,E2 -19941.794} C_VEL
LIN {X 0,Y 261.999,Z 876.286,A -85,B 0,C 180,E1 -19943.833,E2 -19943.833} C_VEL
LIN {X 0,Y 262.571,Z 878.244,A -85,B 0,C 180,E1 -19946.077,E2 -19946.077} C_VEL
LIN {X 0,Y 262.469,Z 880.508,A -85,B 0,C 180,E1 -19947.62,E2 -19947.62} C_VEL
LIN {X 0,Y 261.853,Z 885.173,A -85,B 0,C 180,E1 -19950.197,E2 -19950.197} C_VEL
LIN {X 0,Y 261.349,Z 887.117,A -85,B 0,C 180,E1 -19951.05,E2 -19951.05} C_VEL
LIN {X 0,Y 256.596,Z 894.314,A -85,B 0,C 180,E1 -19953.133,E2 -19953.133} C_VEL
LIN {X 0,Y 252.16,Z 900.21,A -85,B 0,C 180,E1 -19955.287,E2 -19955.287} C_VEL
LIN {X 0,Y 248.05,Z 905.041,A -85,B 0,C 180,E1 -19957.512,E2 -19957.512} C_VEL
LIN {X 0,Y 243.262,Z 909.964,A -85,B 0,C 180,E1 -19960.595,E2 -19960.595} C_VEL
LIN {X 0,Y 239.993,Z 912.487,A -85,B 0,C 180,E1 -19962.972,E2 -19962.972} C_VEL
LIN {X 0,Y 238.06,Z 913.795,A -85,B 0,C 180,E1 -19964.592,E2 -19964.592} C_VEL
LIN {X 0,Y 234.67,Z 915.111,A -85,B 0,C 180,E1 -19967.899,E2 -19967.899} C_VEL
LIN {X 0,Y 233.222,Z 915.325,A -85,B 0,C 180,E1 -19969.583,E2 -19969.583} C_VEL
LIN {X 0,Y 231.05,Z 914.381,A -85,B 0,C 180,E1 -19973.012,E2 -19973.012} C_VEL
LIN {X 0,Y 230.301,Z 913.347,A -85,B 0,C 180,E1 -19974.747,E2 -19974.747} C_VEL
LIN {X 0,Y 229.006,Z 910.06,A -85,B 0,C 180,E1 -19978.241,E2 -19978.241} C_VEL
LIN {X 0,Y 228.306,Z 906.572,A -85,B 0,C 180,E1 -19980.882,E2 -19980.882} C_VEL
LIN {X 0,Y 227.987,Z 902.074,A -85,B 0,C 180,E1 -19983.535,E2 -19983.535} C_VEL
LIN {X 0,Y 228.162,Z 896.467,A -85,B 0,C 180,E1 -19986.189,E2 -19986.189} C_VEL
LIN {X 0,Y 228.58,Z 890.897,A -85,B 0,C 180,E1 -19988.398,E2 -19988.398} C_VEL
LIN {X 0,Y 229.121,Z 883.082,A -85,B 0,C 180,E1 -19991.008,E2 -19991.008} C_VEL
LIN {X 0,Y 229.882,Z 874.865,A -85,B 0,C 180,E1 -19993.255,E2 -19993.255} C_VEL
LIN {X 0,Y 230.8,Z 865.427,A -85,B 0,C 180,E1 -19995.453,E2 -19995.453} C_VEL
LIN {X 0,Y 231.751,Z 855.338,A -85,B 0,C 180,E1 -19997.426,E2 -19997.426} C_VEL
LIN {X 0,Y 232.788,Z 844.677,A -85,B 0,C 180,E1 -19999.167,E2 -19999.167} C_VEL
LIN {X 0,Y 229.697,Z 831.779,A -85,B 0,C 180,E1 -20001.023,E2 -20001.023} C_VEL
LIN {X 0,Y 227.933,Z 824.08,A -85,B 0,C 180,E1 -20002.01,E2 -20002.01} C_VEL
LIN {X 0,Y 227.878,Z 824.087,A -85,B 0,C 180,E1 -20006.564,E2 -20006.564} C_VEL
LIN {X 0,Y 227.878,Z 824.096,A -85,B 0,C 180,E1 -20010.278,E2 -20010.278} C_VEL
LIN {X 0,Y 227.884,Z 824.086,A -85,B 0,C 180,E1 -20013.72,E2 -20013.72} C_VEL
LIN {X 0,Y 227.848,Z 824.092,A -85,B 0,C 180,E1 -20018.091,E2 -20018.091} C_VEL
LIN {X 0,Y 227.793,Z 824.102,A -85,B 0,C 180,E1 -20022.747,E2 -20022.747} C_VEL
LIN {X 0,Y 227.791,Z 824.108,A -85,B 0,C 180,E1 -20027.25,E2 -20027.25} C_VEL
LIN {X 0,Y 227.846,Z 824.104,A -85,B 0,C 180,E1 -20031.906,E2 -20031.906} C_VEL
LIN {X 0,Y 227.886,Z 824.097,A -85,B 0,C 180,E1 -20036.376,E2 -20036.376} C_VEL
LIN {X 0,Y 227.917,Z 824.097,A -85,B 0,C 180,E1 -20038.027,E2 -20038.027} C_VEL
LIN {X 0,Y 228.951,Z 826.999,A -85,B 0,C 180,E1 -20038.457,E2 -20038.457} C_VEL
LIN {X 0,Y 232.185,Z 833.587,A -85,B 0,C 180,E1 -20039.662,E2 -20039.662} C_VEL
LIN {X 0,Y 236.422,Z 843.657,A -85,B 0,C 180,E1 -20041.597,E2 -20041.597} C_VEL
LIN {X 0,Y 239.646,Z 853.773,A -85,B 0,C 180,E1 -20043.666,E2 -20043.666} C_VEL
LIN {X 0,Y 241.731,Z 862.768,A -85,B 0,C 180,E1 -20045.676,E2 -20045.676} C_VEL
LIN {X 0,Y 239.639,Z 872.327,A -85,B 0,C 180,E1 -20047.586,E2 -20047.586} C_VEL
LIN {X 0,Y 237.661,Z 880.672,A -85,B 0,C 180,E1 -20049.665,E2 -20049.665} C_VEL
LIN {X 0,Y 235.728,Z 887.584,A -85,B 0,C 180,E1 -20051.754,E2 -20051.754} C_VEL
LIN {X 0,Y 233.873,Z 894.31,A -85,B 0,C 180,E1 -20054.306,E2 -20054.306} C_VEL
LIN {X 0,Y 232.347,Z 899.682,A -85,B 0,C 180,E1 -20056.885,E2 -20056.885} C_VEL
LIN {X 0,Y 230.734,Z 903.948,A -85,B 0,C 180,E1 -20059.467,E2 -20059.467} C_VEL
LIN {X 0,Y 230.031,Z 906.174,A -85,B 0,C 180,E1 -20061.21,E2 -20061.21} C_VEL
LIN {X 0,Y 229.535,Z 907.975,A -85,B 0,C 180,E1 -20062.962,E2 -20062.962} C_VEL
LIN {X 0,Y 229.255,Z 909.314,A -85,B 0,C 180,E1 -20064.72,E2 -20064.72} C_VEL
LIN {X 0,Y 228.672,Z 910.892,A -85,B 0,C 180,E1 -20068.236,E2 -20068.236} C_VEL
LIN {X 0,Y 228.592,Z 911.12,A -85,B 0,C 180,E1 -20069.997,E2 -20069.997} C_VEL
LIN {X 0,Y 228.918,Z 910.349,A -85,B 0,C 180,E1 -20073.517,E2 -20073.517} C_VEL
LIN {X 0,Y 229.235,Z 909.404,A -85,B 0,C 180,E1 -20075.274,E2 -20075.274} C_VEL
LIN {X 0,Y 229.431,Z 908.115,A -85,B 0,C 180,E1 -20077.035,E2 -20077.035} C_VEL
LIN {X 0,Y 230.356,Z 905.306,A -85,B 0,C 180,E1 -20079.657,E2 -20079.657} C_VEL
LIN {X 0,Y 231.816,Z 901.458,A -85,B 0,C 180,E1 -20082.249,E2 -20082.249} C_VEL
LIN {X 0,Y 233.34,Z 896.542,A -85,B 0,C 180,E1 -20084.83,E2 -20084.83} C_VEL
LIN {X 0,Y 235.016,Z 890.36,A -85,B 0,C 180,E1 -20087.397,E2 -20087.397} C_VEL
LIN {X 0,Y 237.162,Z 882.584,A -85,B 0,C 180,E1 -20089.921,E2 -20089.921} C_VEL
LIN {X 0,Y 239.177,Z 874.645,A -85,B 0,C 180,E1 -20091.999,E2 -20091.999} C_VEL
LIN {X 0,Y 241.4,Z 864.938,A -85,B 0,C 180,E1 -20094.05,E2 -20094.05} C_VEL
LIN {X 0,Y 241.756,Z 862.115,A -85,B 0,C 180,E1 -20094.592,E2 -20094.592} C_VEL
LIN {X 0,Y 239.52,Z 853.279,A -85,B 0,C 180,E1 -20096.577,E2 -20096.577} C_VEL
LIN {X 0,Y 236.238,Z 843.174,A -85,B 0,C 180,E1 -20098.642,E2 -20098.642} C_VEL
LIN {X 0,Y 232.913,Z 835.147,A -85,B 0,C 180,E1 -20100.182,E2 -20100.182} C_VEL
LIN {X 0,Y 228.078,Z 824.924,A -85,B 0,C 180,E1 -20102.018,E2 -20102.018} C_VEL
LIN {X 0,Y 227.898,Z 824.099,A -85,B 0,C 180,E1 -20102.122,E2 -20102.122} C_VEL
LIN {X 0,Y 227.902,Z 824.099,A -85,B 0,C 180,E1 -20106.699,E2 -20106.699} C_VEL
LIN {X 0,Y 227.896,Z 824.099,A -85,B 0,C 180,E1 -20110.357,E2 -20110.357} C_VEL
LIN {X 0,Y 227.911,Z 824.096,A -85,B 0,C 180,E1 -20114.827,E2 -20114.827} C_VEL
LIN {X 0,Y 227.93,Z 824.086,A -85,B 0,C 180,E1 -20117.727,E2 -20117.727} C_VEL
LIN {X 0,Y 227.88,Z 824.092,A -85,B 0,C 180,E1 -20121.916,E2 -20121.916} C_VEL
LIN {X 0,Y 227.878,Z 824.093,A -85,B 0,C 180,E1 -20126.371,E2 -20126.371} C_VEL
LIN {X 0,Y 227.907,Z 824.088,A -85,B 0,C 180,E1 -20130.436,E2 -20130.436} C_VEL
LIN {X 0,Y 227.916,Z 824.088,A -85,B 0,C 180,E1 -20134.424,E2 -20134.424} C_VEL
LIN {X 0,Y 227.949,Z 824.088,A -85,B 0,C 180,E1 -20138.286,E2 -20138.286} C_VEL
LIN {X 0,Y 228.021,Z 824.079,A -85,B 0,C 180,E1 -20142.825,E2 -20142.825} C_VEL
LIN {X 0,Y 228.08,Z 824.078,A -85,B 0,C 180,E1 -20147.543,E2 -20147.543} C_VEL
LIN {X 0,Y 228.29,Z 824.039,A -85,B 0,C 180,E1 -20151.145,E2 -20151.145} C_VEL
LIN {X 0,Y 228.338,Z 824.044,A -85,B 0,C 180,E1 -20152.928,E2 -20152.928} C_VEL
LIN {X 0,Y 228.539,Z 824.018,A -85,B 0,C 180,E1 -20158.238,E2 -20158.238} C_VEL
LIN {X 0,Y 228.538,Z 824.022,A -85,B 0,C 180,E1 -20161.762,E2 -20161.762} C_VEL
LIN {X 0,Y 228.334,Z 824.042,A -85,B 0,C 180,E1 -20167.072,E2 -20167.072} C_VEL
LIN {X 0,Y 228.144,Z 824.065,A -85,B 0,C 180,E1 -20170.651,E2 -20170.651} C_VEL
LIN {X 0,Y 228.05,Z 824.08,A -85,B 0,C 180,E1 -20174.273,E2 -20174.273} C_VEL
LIN {X 0,Y 227.988,Z 824.087,A -85,B 0,C 180,E1 -20177.954,E2 -20177.954} C_VEL
LIN {X 0,Y 227.907,Z 824.099,A -85,B 0,C 180,E1 -20182.325,E2 -20182.325} C_VEL
LIN {X 0,Y 227.908,Z 824.093,A -85,B 0,C 180,E1 -20186.594,E2 -20186.594} C_VEL
LIN {X 0,Y 227.865,Z 824.159,A -85,B 0,C 180,E1 -20191.054,E2 -20191.054} C_VEL
LIN {X 0,Y 229.167,Z 829.913,A -85,B 0,C 180,E1 -20195.64,E2 -20195.64} C_VEL
LIN {X 0,Y 230.443,Z 836.442,A -85,B 0,C 180,E1 -20200.326,E2 -20200.326} C_VEL
LIN {X 0,Y 231.852,Z 843.558,A -85,B 0,C 180,E1 -20205.057,E2 -20205.057} C_VEL
LIN {X 0,Y 232.965,Z 849.846,A -85,B 0,C 180,E1 -20208.955,E2 -20208.955} C_VEL
LIN {X 0,Y 233.197,Z 852.865,A -85,B 0,C 180,E1 -20210.741,E2 -20210.741} C_VEL
LIN {X 0,Y 231.832,Z 858.558,A -85,B 0,C 180,E1 -20213.864,E2 -20213.864} C_VEL
LIN {X 0,Y 231.243,Z 860.538,A -85,B 0,C 180,E1 -20214.673,E2 -20214.673} C_VEL
LIN {X 0,Y 229.997,Z 864.565,A -85,B 0,C 180,E1 -20215.676,E2 -20215.676} C_VEL
LIN {X 0,Y 228.238,Z 871.119,A -85,B 0,C 180,E1 -20216.7,E2 -20216.7} C_VEL
LIN {X 0,Y 227.26,Z 876.593,A -85,B 0,C 180,E1 -20217.328,E2 -20217.328} C_VEL
LIN {X 0,Y 227.03,Z 882.21,A -85,B 0,C 180,E1 -20217.907,E2 -20217.907} C_VEL
LIN {X 0,Y 227.196,Z 884.076,A -85,B 0,C 180,E1 -20218.1,E2 -20218.1} C_VEL
LIN {X 0,Y 228.29,Z 896.64,A -85,B 0,C 180,E1 -20219.541,E2 -20219.541} C_VEL
LIN {X 0,Y 228.641,Z 907.708,A -85,B 0,C 180,E1 -20221.049,E2 -20221.049} C_VEL
LIN {X 0,Y 228.325,Z 918.575,A -85,B 0,C 180,E1 -20222.786,E2 -20222.786} C_VEL
LIN {X 0,Y 227.54,Z 928.342,A -85,B 0,C 180,E1 -20224.628,E2 -20224.628} C_VEL
LIN {X 0,Y 226.359,Z 937.543,A -85,B 0,C 180,E1 -20226.684,E2 -20226.684} C_VEL
LIN {X 0,Y 225.617,Z 942.827,A -85,B 0,C 180,E1 -20228.054,E2 -20228.054} C_VEL
LIN {X 0,Y 223.603,Z 950.575,A -85,B 0,C 180,E1 -20230.354,E2 -20230.354} C_VEL
LIN {X 0,Y 221.937,Z 956.506,A -85,B 0,C 180,E1 -20232.496,E2 -20232.496} C_VEL
LIN {X 0,Y 220.766,Z 962.716,A -85,B 0,C 180,E1 -20235.249,E2 -20235.249} C_VEL
LIN {X 0,Y 219.996,Z 967.662,A -85,B 0,C 180,E1 -20238.019,E2 -20238.019} C_VEL
LIN {X 0,Y 219.744,Z 971.501,A -85,B 0,C 180,E1 -20240.802,E2 -20240.802} C_VEL
LIN {X 0,Y 219.829,Z 973.511,A -85,B 0,C 180,E1 -20242.656,E2 -20242.656} C_VEL
LIN {X 0,Y 220.045,Z 975.042,A -85,B 0,C 180,E1 -20244.505,E2 -20244.505} C_VEL
LIN {X 0,Y 220.304,Z 976.148,A -85,B 0,C 180,E1 -20246.345,E2 -20246.345} C_VEL
LIN {X 0,Y 220.538,Z 976.832,A -85,B 0,C 180,E1 -20248.177,E2 -20248.177} C_VEL
LIN {X 0,Y 220.779,Z 977.093,A -85,B 0,C 180,E1 -20250.003,E2 -20250.003} C_VEL
LIN {X 0,Y 220.542,Z 976.821,A -85,B 0,C 180,E1 -20251.829,E2 -20251.829} C_VEL
LIN {X 0,Y 220.316,Z 976.13,A -85,B 0,C 180,E1 -20253.661,E2 -20253.661} C_VEL
LIN {X 0,Y 220.07,Z 975.016,A -85,B 0,C 180,E1 -20255.501,E2 -20255.501} C_VEL
LIN {X 0,Y 219.831,Z 973.151,A -85,B 0,C 180,E1 -20257.661,E2 -20257.661} C_VEL
LIN {X 0,Y 219.888,Z 969.585,A -85,B 0,C 180,E1 -20261.059,E2 -20261.059} C_VEL
LIN {X 0,Y 220.746,Z 966.481,A -85,B 0,C 180,E1 -20264.759,E2 -20264.759} C_VEL
LIN {X 0,Y 222.768,Z 962.118,A -85,B 0,C 180,E1 -20268.393,E2 -20268.393} C_VEL
LIN {X 0,Y 225.952,Z 956.327,A -85,B 0,C 180,E1 -20271.919,E2 -20271.919} C_VEL
LIN {X 0,Y 230.249,Z 948.95,A -85,B 0,C 180,E1 -20275.301,E2 -20275.301} C_VEL
LIN {X 0,Y 233.999,Z 941.328,A -85,B 0,C 180,E1 -20278.235,E2 -20278.235} C_VEL
LIN {X 0,Y 237.967,Z 933.701,A -85,B 0,C 180,E1 -20280.688,E2 -20280.688} C_VEL
LIN {X 0,Y 241.027,Z 927.375,A -85,B 0,C 180,E1 -20282.549,E2 -20282.549} C_VEL
LIN {X 0,Y 244.977,Z 916.894,A -85,B 0,C 180,E1 -20285.556,E2 -20285.556} C_VEL
LIN {X 0,Y 248.41,Z 906.632,A -85,B 0,C 180,E1 -20288.496,E2 -20288.496} C_VEL
LIN {X 0,Y 251.515,Z 896.915,A -85,B 0,C 180,E1 -20291.413,E2 -20291.413} C_VEL
LIN {X 0,Y 253.939,Z 889.858,A -85,B 0,C 180,E1 -20293.784,E2 -20293.784} C_VEL
LIN {X 0,Y 254.704,Z 887.504,A -85,B 0,C 180,E1 -20294.743,E2 -20294.743} C_VEL
LIN {X 0,Y 255.22,Z 885.687,A -85,B 0,C 180,E1 -20295.725,E2 -20295.725} C_VEL
LIN {X 0,Y 255.965,Z 883.068,A -85,B 0,C 180,E1 -20297.849,E2 -20297.849} C_VEL
LIN {X 0,Y 256.637,Z 881.674,A -85,B 0,C 180,E1 -20300.069,E2 -20300.069} C_VEL
LIN {X 0,Y 257.334,Z 881.503,A -85,B 0,C 180,E1 -20302.377,E2 -20302.377} C_VEL
LIN {X 0,Y 257.75,Z 882.704,A -85,B 0,C 180,E1 -20304.889,E2 -20304.889} C_VEL
LIN {X 0,Y 257.871,Z 883.887,A -85,B 0,C 180,E1 -20306.137,E2 -20306.137} C_VEL
LIN {X 0,Y 257.132,Z 887.729,A -85,B 0,C 180,E1 -20308.714,E2 -20308.714} C_VEL
LIN {X 0,Y 256.784,Z 889.234,A -85,B 0,C 180,E1 -20309.547,E2 -20309.547} C_VEL
LIN {X 0,Y 255.904,Z 891.134,A -85,B 0,C 180,E1 -20310.374,E2 -20310.374} C_VEL
LIN {X 0,Y 250.882,Z 897.769,A -85,B 0,C 180,E1 -20312.47,E2 -20312.47} C_VEL
LIN {X 0,Y 246.257,Z 903.268,A -85,B 0,C 180,E1 -20314.654,E2 -20314.654} C_VEL
LIN {X 0,Y 241.957,Z 907.754,A -85,B 0,C 180,E1 -20316.913,E2 -20316.913} C_VEL
LIN {X 0,Y 238.14,Z 911.336,A -85,B 0,C 180,E1 -20319.259,E2 -20319.259} C_VEL
LIN {X 0,Y 233.505,Z 914.573,A -85,B 0,C 180,E1 -20322.484,E2 -20322.484} C_VEL
LIN {X 0,Y 229.64,Z 916.405,A -85,B 0,C 180,E1 -20325.828,E2 -20325.828} C_VEL
LIN {X 0,Y 226.389,Z 916.693,A -85,B 0,C 180,E1 -20329.265,E2 -20329.265} C_VEL
LIN {X 0,Y 224.095,Z 915.478,A -85,B 0,C 180,E1 -20332.794,E2 -20332.794} C_VEL
LIN {X 0,Y 222.557,Z 912.654,A -85,B 0,C 180,E1 -20336.379,E2 -20336.379} C_VEL
LIN {X 0,Y 221.31,Z 908.361,A -85,B 0,C 180,E1 -20340,E2 -20340} C_VEL
LIN {X 0,Y 221.064,Z 903.966,A -85,B 0,C 180,E1 -20342.733,E2 -20342.733} C_VEL
LIN {X 0,Y 221.04,Z 897.42,A -85,B 0,C 180,E1 -20345.931,E2 -20345.931} C_VEL
LIN {X 0,Y 221.46,Z 891.66,A -85,B 0,C 180,E1 -20348.261,E2 -20348.261} C_VEL
LIN {X 0,Y 222.007,Z 883.81,A -85,B 0,C 180,E1 -20350.949,E2 -20350.949} C_VEL
LIN {X 0,Y 222.754,Z 875.68,A -85,B 0,C 180,E1 -20353.223,E2 -20353.223} C_VEL
LIN {X 0,Y 223.55,Z 867.212,A -85,B 0,C 180,E1 -20355.266,E2 -20355.266} C_VEL
LIN {X 0,Y 224.408,Z 858.441,A -85,B 0,C 180,E1 -20357.074,E2 -20357.074} C_VEL
LIN {X 0,Y 225.435,Z 848.319,A -85,B 0,C 180,E1 -20358.861,E2 -20358.861} C_VEL
LIN {X 0,Y 225.697,Z 845.493,A -85,B 0,C 180,E1 -20359.303,E2 -20359.303} C_VEL
LIN {X 0,Y 222.623,Z 832.648,A -85,B 0,C 180,E1 -20361.197,E2 -20361.197} C_VEL
LIN {X 0,Y 220.882,Z 824.959,A -85,B 0,C 180,E1 -20362.2,E2 -20362.2} C_VEL
LIN {X 0,Y 220.835,Z 824.962,A -85,B 0,C 180,E1 -20366.984,E2 -20366.984} C_VEL
LIN {X 0,Y 220.827,Z 824.973,A -85,B 0,C 180,E1 -20370.758,E2 -20370.758} C_VEL
LIN {X 0,Y 220.801,Z 824.977,A -85,B 0,C 180,E1 -20374.955,E2 -20374.955} C_VEL
LIN {X 0,Y 220.81,Z 824.969,A -85,B 0,C 180,E1 -20377.274,E2 -20377.274} C_VEL
LIN {X 0,Y 220.756,Z 824.978,A -85,B 0,C 180,E1 -20381.956,E2 -20381.956} C_VEL
LIN {X 0,Y 220.76,Z 824.982,A -85,B 0,C 180,E1 -20385.539,E2 -20385.539} C_VEL
LIN {X 0,Y 220.787,Z 824.979,A -85,B 0,C 180,E1 -20390.455,E2 -20390.455} C_VEL
LIN {X 0,Y 220.832,Z 824.972,A -85,B 0,C 180,E1 -20392.791,E2 -20392.791} C_VEL
LIN {X 0,Y 220.874,Z 824.969,A -85,B 0,C 180,E1 -20396.813,E2 -20396.813} C_VEL
LIN {X 0,Y 221.866,Z 827.728,A -85,B 0,C 180,E1 -20397.281,E2 -20397.281} C_VEL
LIN {X 0,Y 226.93,Z 838.243,A -85,B 0,C 180,E1 -20399.328,E2 -20399.328} C_VEL
LIN {X 0,Y 230.552,Z 847.24,A -85,B 0,C 180,E1 -20401.188,E2 -20401.188} C_VEL
LIN {X 0,Y 233.566,Z 857.291,A -85,B 0,C 180,E1 -20403.381,E2 -20403.381} C_VEL
LIN {X 0,Y 235.05,Z 863.622,A -85,B 0,C 180,E1 -20404.889,E2 -20404.889} C_VEL
LIN {X 0,Y 234.824,Z 866.376,A -85,B 0,C 180,E1 -20405.461,E2 -20405.461} C_VEL
LIN {X 0,Y 232.784,Z 875.132,A -85,B 0,C 180,E1 -20407.357,E2 -20407.357} C_VEL
LIN {X 0,Y 230.63,Z 883.167,A -85,B 0,C 180,E1 -20409.483,E2 -20409.483} C_VEL
LIN {X 0,Y 228.756,Z 889.813,A -85,B 0,C 180,E1 -20411.642,E2 -20411.642} C_VEL
LIN {X 0,Y 227.118,Z 895.343,A -85,B 0,C 180,E1 -20413.826,E2 -20413.826} C_VEL
LIN {X 0,Y 225.512,Z 900.715,A -85,B 0,C 180,E1 -20416.48,E2 -20416.48} C_VEL
LIN {X 0,Y 223.832,Z 904.98,A -85,B 0,C 180,E1 -20419.138,E2 -20419.138} C_VEL
LIN {X 0,Y 223.091,Z 907.206,A -85,B 0,C 180,E1 -20420.934,E2 -20420.934} C_VEL
LIN {X 0,Y 222.58,Z 909.005,A -85,B 0,C 180,E1 -20422.741,E2 -20422.741} C_VEL
LIN {X 0,Y 222.265,Z 910.346,A -85,B 0,C 180,E1 -20424.554,E2 -20424.554} C_VEL
LIN {X 0,Y 221.652,Z 911.924,A -85,B 0,C 180,E1 -20428.18,E2 -20428.18} C_VEL
LIN {X 0,Y 221.568,Z 912.152,A -85,B 0,C 180,E1 -20429.997,E2 -20429.997} C_VEL
LIN {X 0,Y 221.907,Z 911.379,A -85,B 0,C 180,E1 -20433.628,E2 -20433.628} C_VEL
LIN {X 0,Y 222.24,Z 910.435,A -85,B 0,C 180,E1 -20435.441,E2 -20435.441} C_VEL
LIN {X 0,Y 222.46,Z 909.145,A -85,B 0,C 180,E1 -20437.256,E2 -20437.256} C_VEL
LIN {X 0,Y 223.433,Z 906.336,A -85,B 0,C 180,E1 -20439.959,E2 -20439.959} C_VEL
LIN {X 0,Y 224.956,Z 902.489,A -85,B 0,C 180,E1 -20442.629,E2 -20442.629} C_VEL
LIN {X 0,Y 226.556,Z 897.571,A -85,B 0,C 180,E1 -20445.285,E2 -20445.285} C_VEL
LIN {X 0,Y 228.322,Z 891.389,A -85,B 0,C 180,E1 -20447.924,E2 -20447.924} C_VEL
LIN {X 0,Y 230.57,Z 883.613,A -85,B 0,C 180,E1 -20450.516,E2 -20450.516} C_VEL
LIN {X 0,Y 232.678,Z 875.673,A -85,B 0,C 180,E1 -20452.647,E2 -20452.647} C_VEL
LIN {X 0,Y 235.004,Z 865.965,A -85,B 0,C 180,E1 -20454.748,E2 -20454.748} C_VEL
LIN {X 0,Y 235.256,Z 864.575,A -85,B 0,C 180,E1 -20455.018,E2 -20455.018} C_VEL
LIN {X 0,Y 233.517,Z 856.961,A -85,B 0,C 180,E1 -20456.833,E2 -20456.833} C_VEL
LIN {X 0,Y 230.697,Z 847.768,A -85,B 0,C 180,E1 -20458.854,E2 -20458.854} C_VEL
LIN {X 0,Y 227.319,Z 839.114,A -85,B 0,C 180,E1 -20460.64,E2 -20460.64} C_VEL
LIN {X 0,Y 222.671,Z 829.068,A -85,B 0,C 180,E1 -20462.599,E2 -20462.599} C_VEL
LIN {X 0,Y 221.04,Z 825.93,A -85,B 0,C 180,E1 -20463.186,E2 -20463.186} C_VEL
LIN {X 0,Y 220.843,Z 824.977,A -85,B 0,C 180,E1 -20463.314,E2 -20463.314} C_VEL
LIN {X 0,Y 220.831,Z 824.979,A -85,B 0,C 180,E1 -20467.285,E2 -20467.285} C_VEL
LIN {X 0,Y 220.866,Z 824.975,A -85,B 0,C 180,E1 -20471.925,E2 -20471.925} C_VEL
LIN {X 0,Y 220.866,Z 824.973,A -85,B 0,C 180,E1 -20475.569,E2 -20475.569} C_VEL
LIN {X 0,Y 220.868,Z 824.973,A -85,B 0,C 180,E1 -20479.784,E2 -20479.784} C_VEL
LIN {X 0,Y 220.833,Z 824.976,A -85,B 0,C 180,E1 -20482.794,E2 -20482.794} C_VEL
LIN {X 0,Y 220.813,Z 824.979,A -85,B 0,C 180,E1 -20487.243,E2 -20487.243} C_VEL
LIN {X 0,Y 220.824,Z 824.977,A -85,B 0,C 180,E1 -20491.485,E2 -20491.485} C_VEL
LIN {X 0,Y 220.854,Z 824.971,A -85,B 0,C 180,E1 -20495.563,E2 -20495.563} C_VEL
LIN {X 0,Y 220.879,Z 824.964,A -85,B 0,C 180,E1 -20499.512,E2 -20499.512} C_VEL
LIN {X 0,Y 221.002,Z 824.948,A -85,B 0,C 180,E1 -20503.369,E2 -20503.369} C_VEL
LIN {X 0,Y 221.098,Z 824.944,A -85,B 0,C 180,E1 -20509.005,E2 -20509.005} C_VEL
LIN {X 0,Y 221.273,Z 824.923,A -85,B 0,C 180,E1 -20512.701,E2 -20512.701} C_VEL
LIN {X 0,Y 221.497,Z 824.894,A -85,B 0,C 180,E1 -20518.182,E2 -20518.182} C_VEL
LIN {X 0,Y 221.496,Z 824.9,A -85,B 0,C 180,E1 -20521.818,E2 -20521.818} C_VEL
LIN {X 0,Y 221.27,Z 824.923,A -85,B 0,C 180,E1 -20527.299,E2 -20527.299} C_VEL
LIN {X 0,Y 221.092,Z 824.944,A -85,B 0,C 180,E1 -20530.995,E2 -20530.995} C_VEL
LIN {X 0,Y 221.002,Z 824.958,A -85,B 0,C 180,E1 -20536.631,E2 -20536.631} C_VEL
LIN {X 0,Y 220.872,Z 824.976,A -85,B 0,C 180,E1 -20540.488,E2 -20540.488} C_VEL
LIN {X 0,Y 220.833,Z 824.978,A -85,B 0,C 180,E1 -20544.439,E2 -20544.439} C_VEL
LIN {X 0,Y 220.79,Z 824.981,A -85,B 0,C 180,E1 -20548.52,E2 -20548.52} C_VEL
LIN {X 0,Y 220.857,Z 825.101,A -85,B 0,C 180,E1 -20550.079,E2 -20550.079} C_VEL
LIN {X 0,Y 222.085,Z 830.659,A -85,B 0,C 180,E1 -20554.724,E2 -20554.724} C_VEL
LIN {X 0,Y 223.219,Z 836.343,A -85,B 0,C 180,E1 -20559.028,E2 -20559.028} C_VEL
LIN {X 0,Y 224.446,Z 842.776,A -85,B 0,C 180,E1 -20563.542,E2 -20563.542} C_VEL
LIN {X 0,Y 225.569,Z 848.667,A -85,B 0,C 180,E1 -20567.395,E2 -20567.395} C_VEL
LIN {X 0,Y 226.22,Z 853.302,A -85,B 0,C 180,E1 -20570.283,E2 -20570.283} C_VEL
LIN {X 0,Y 224.397,Z 860.756,A -85,B 0,C 180,E1 -20574.519,E2 -20574.519} C_VEL
LIN {X 0,Y 223.653,Z 863.766,A -85,B 0,C 180,E1 -20576.218,E2 -20576.218} C_VEL
LIN {X 0,Y 226.44,Z 878.572,A -85,B 0,C 180,E1 -20577.536,E2 -20577.536} C_VEL
LIN {X 0,Y 227.196,Z 884.076,A -85,B 0,C 180,E1 -20578.1,E2 -20578.1} C_VEL
LIN {X 0,Y 227.196,Z 889.632,A -85,B 0,C 180,E1 -20578.628,E2 -20578.628} C_VEL
LIN {X 0,Y 226.177,Z 895.201,A -85,B 0,C 180,E1 -20579.098,E2 -20579.098} C_VEL
